Yaskawa INFORM job: DEMO_ROOF_SIDE_0625_3PAINT_40.JBI

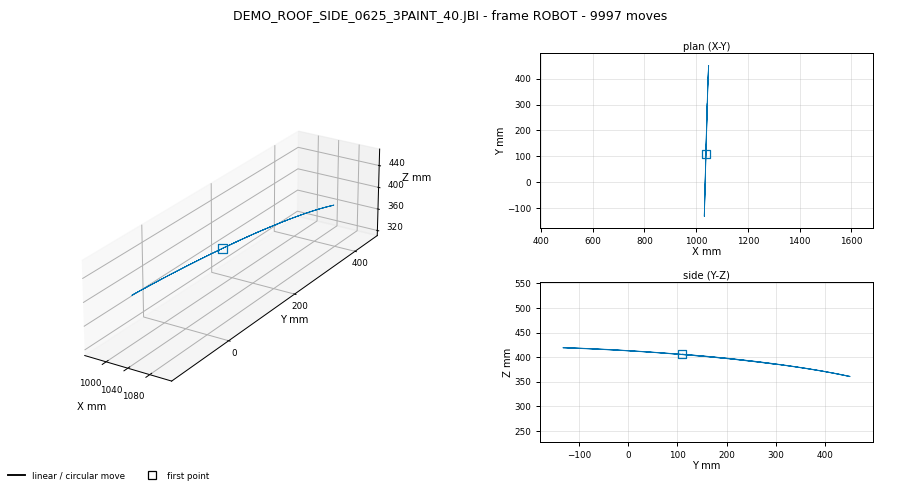
[picture p0: tool path of DEMO_ROOF_SIDE_0625_3PAINT_40.JBI in frame ROBOT, 9997 of 9997 moves have a stored position in this frame; points joined in program order, loops and branches not executed]
/JOB
//NAME DEMO_ROOF_SIDE_0625_3PAINT40
//POS
///NPOS 9997,0,0,0,0,0
///TOOL 0
///USER 0
///POSTYPE ROBOT
///RECTAN
///RCONF 1,0,0,0,0,0,0,0,0,0,0,0,0,0,0,0,0,0,0,0,0,0,0,0
C00000=1038.279,110.254,406.357,169.691,40.048,157.539
C00001=1038.285,110.504,406.337,169.693,40.048,157.539
C00002=1038.291,110.753,406.317,169.696,40.048,157.539
C00003=1038.297,111.002,406.297,169.698,40.048,157.539
C00004=1038.304,111.251,406.277,169.700,40.048,157.539
C00005=1038.310,111.500,406.257,169.702,40.049,157.539
C00006=1038.316,111.749,406.238,169.704,40.049,157.539
C00007=1038.323,111.998,406.218,169.706,40.049,157.539
C00008=1038.329,112.248,406.198,169.708,40.050,157.540
C00009=1038.335,112.497,406.178,169.710,40.049,157.540
C00010=1038.341,112.746,406.158,169.713,40.050,157.540
C00011=1038.347,112.995,406.138,169.715,40.050,157.540
C00012=1038.354,113.244,406.118,169.717,40.050,157.540
C00013=1038.359,113.494,406.097,169.719,40.051,157.540
C00014=1038.365,113.742,406.077,169.721,40.051,157.540
C00015=1038.372,113.992,406.057,169.723,40.051,157.540
C00016=1038.378,114.241,406.037,169.725,40.051,157.541
C00017=1038.383,114.490,406.016,169.727,40.052,157.541
C00018=1038.390,114.739,405.996,169.730,40.052,157.541
C00019=1038.396,114.988,405.976,169.732,40.052,157.541
C00020=1038.402,115.237,405.956,169.734,40.052,157.541
C00021=1038.407,115.487,405.935,169.736,40.053,157.541
C00022=1038.414,115.735,405.915,169.738,40.053,157.542
C00023=1038.420,115.984,405.895,169.740,40.053,157.542
C00024=1038.426,116.233,405.874,169.742,40.054,157.542
C00025=1038.432,116.482,405.854,169.745,40.054,157.542
C00026=1038.438,116.732,405.833,169.747,40.054,157.542
C00027=1038.444,116.981,405.813,169.749,40.054,157.542
C00028=1038.450,117.230,405.793,169.751,40.055,157.542
C00029=1038.456,117.479,405.773,169.753,40.055,157.543
C00030=1038.462,117.728,405.753,169.755,40.056,157.543
C00031=1038.469,117.977,405.732,169.757,40.055,157.543
C00032=1038.474,118.226,405.711,169.759,40.056,157.543
C00033=1038.480,118.475,405.691,169.762,40.056,157.543
C00034=1038.487,118.725,405.671,169.765,40.057,157.543
C00035=1038.493,118.973,405.651,169.767,40.057,157.543
C00036=1038.499,119.223,405.630,169.769,40.057,157.544
C00037=1038.505,119.471,405.609,169.771,40.057,157.544
C00038=1038.511,119.721,405.589,169.773,40.058,157.544
C00039=1038.517,119.970,405.569,169.775,40.058,157.544
C00040=1038.523,120.219,405.548,169.777,40.058,157.544
C00041=1038.529,120.468,405.528,169.780,40.059,157.544
C00042=1038.536,120.716,405.507,169.782,40.059,157.544
C00043=1038.541,120.966,405.486,169.784,40.059,157.544
C00044=1038.547,121.215,405.466,169.786,40.059,157.545
C00045=1038.554,121.465,405.446,169.788,40.060,157.545
C00046=1038.560,121.713,405.425,169.790,40.060,157.545
C00047=1038.566,121.963,405.404,169.792,40.060,157.545
C00048=1038.572,122.211,405.385,169.794,40.060,157.545
C00049=1038.579,122.460,405.363,169.797,40.061,157.545
C00050=1038.584,122.710,405.343,169.800,40.061,157.545
C00051=1038.591,122.959,405.323,169.802,40.061,157.546
C00052=1038.597,123.208,405.303,169.804,40.062,157.546
C00053=1038.603,123.457,405.281,169.806,40.061,157.546
C00054=1038.609,123.706,405.261,169.808,40.062,157.546
C00055=1038.616,123.955,405.241,169.810,40.062,157.546
C00056=1038.621,124.204,405.219,169.812,40.063,157.546
C00057=1038.628,124.453,405.199,169.814,40.062,157.546
C00058=1038.635,124.739,405.175,169.818,40.063,157.547
C00059=1038.642,125.025,405.151,169.820,40.063,157.547
C00060=1038.649,125.311,405.129,169.822,40.064,157.547
C00061=1038.656,125.596,405.105,169.825,40.064,157.547
C00062=1038.663,125.845,405.084,169.827,40.064,157.547
C00063=1038.668,126.094,405.063,169.829,40.064,157.547
C00064=1038.675,126.344,405.043,169.831,40.065,157.548
C00065=1038.682,126.593,405.022,169.833,40.065,157.548
C00066=1038.687,126.842,405.001,169.836,40.065,157.548
C00067=1038.694,127.091,404.980,169.838,40.065,157.548
C00068=1038.700,127.340,404.960,169.840,40.065,157.548
C00069=1038.706,127.589,404.939,169.843,40.066,157.548
C00070=1038.713,127.838,404.918,169.845,40.066,157.548
C00071=1038.719,128.086,404.898,169.847,40.067,157.549
C00072=1038.725,128.336,404.877,169.849,40.066,157.549
C00073=1038.731,128.585,404.857,169.851,40.067,157.549
C00074=1038.738,128.834,404.836,169.854,40.067,157.549
C00075=1038.744,129.084,404.815,169.856,40.067,157.549
C00076=1038.750,129.332,404.794,169.858,40.068,157.549
C00077=1038.757,129.582,404.774,169.861,40.068,157.549
C00078=1038.763,129.831,404.752,169.863,40.068,157.549
C00079=1038.769,130.080,404.732,169.865,40.068,157.550
C00080=1038.776,130.328,404.711,169.867,40.069,157.550
C00081=1038.782,130.578,404.690,169.869,40.068,157.550
C00082=1038.788,130.826,404.670,169.872,40.069,157.550
C00083=1038.795,131.075,404.649,169.874,40.069,157.550
C00084=1038.801,131.325,404.628,169.877,40.070,157.550
C00085=1038.806,131.574,404.606,169.879,40.070,157.551
C00086=1038.813,131.823,404.585,169.881,40.070,157.551
C00087=1038.818,132.072,404.565,169.883,40.070,157.551
C00088=1038.824,132.321,404.543,169.885,40.071,157.551
C00089=1038.831,132.570,404.522,169.888,40.071,157.551
C00090=1038.837,132.819,404.502,169.890,40.072,157.551
C00091=1038.843,133.068,404.480,169.892,40.072,157.551
C00092=1038.850,133.317,404.459,169.894,40.073,157.552
C00093=1038.855,133.566,404.438,169.896,40.072,157.552
C00094=1038.861,133.815,404.417,169.899,40.073,157.552
C00095=1038.868,134.064,404.396,169.901,40.073,157.552
C00096=1038.874,134.313,404.374,169.904,40.074,157.552
C00097=1038.879,134.563,404.354,169.906,40.074,157.552
C00098=1038.886,134.811,404.332,169.908,40.075,157.553
C00099=1038.892,135.060,404.311,169.910,40.074,157.553
C00100=1038.898,135.309,404.290,169.912,40.075,157.553
C00101=1038.905,135.559,404.269,169.914,40.075,157.553
C00102=1038.910,135.807,404.248,169.917,40.076,157.553
C00103=1038.916,136.056,404.226,169.920,40.076,157.553
C00104=1038.923,136.305,404.205,169.922,40.076,157.554
C00105=1038.928,136.554,404.185,169.924,40.076,157.554
C00106=1038.935,136.804,404.163,169.926,40.077,157.554
C00107=1038.942,137.053,404.142,169.928,40.077,157.554
C00108=1038.948,137.302,404.120,169.930,40.078,157.554
C00109=1038.953,137.550,404.099,169.933,40.078,157.554
C00110=1038.959,137.799,404.078,169.936,40.078,157.554
C00111=1038.966,138.048,404.056,169.938,40.079,157.555
C00112=1038.972,138.297,404.036,169.940,40.079,157.555
C00113=1038.978,138.547,404.014,169.942,40.079,157.555
C00114=1038.984,138.796,403.993,169.944,40.080,157.555
C00115=1038.991,139.045,403.972,169.947,40.080,157.555
C00116=1038.996,139.293,403.950,169.949,40.080,157.555
C00117=1039.003,139.542,403.929,169.952,40.081,157.556
C00118=1039.009,139.792,403.907,169.954,40.081,157.556
C00119=1039.015,140.041,403.885,169.956,40.082,157.556
C00120=1039.020,140.289,403.864,169.958,40.082,157.556
C00121=1039.027,140.539,403.843,169.960,40.083,157.556
C00122=1039.035,140.824,403.818,169.963,40.083,157.556
C00123=1039.041,141.110,403.794,169.966,40.083,157.557
C00124=1039.048,141.396,403.768,169.969,40.084,157.557
C00125=1039.055,141.681,403.745,169.971,40.084,157.557
C00126=1039.061,141.930,403.723,169.973,40.085,157.557
C00127=1039.067,142.179,403.701,169.976,40.085,157.557
C00128=1039.073,142.428,403.680,169.978,40.085,157.558
C00129=1039.079,142.676,403.658,169.981,40.086,157.558
C00130=1039.085,142.926,403.636,169.983,40.086,157.558
C00131=1039.092,143.175,403.614,169.985,40.087,157.558
C00132=1039.098,143.424,403.593,169.987,40.087,157.558
C00133=1039.103,143.673,403.571,169.990,40.088,157.558
C00134=1039.110,143.922,403.550,169.992,40.088,157.559
C00135=1039.116,144.171,403.528,169.995,40.088,157.559
C00136=1039.122,144.420,403.507,169.997,40.089,157.559
C00137=1039.129,144.669,403.486,169.999,40.089,157.559
C00138=1039.135,144.918,403.464,170.001,40.089,157.559
C00139=1039.141,145.166,403.442,170.004,40.089,157.559
C00140=1039.147,145.415,403.420,170.006,40.090,157.560
C00141=1039.153,145.665,403.399,170.008,40.090,157.560
C00142=1039.159,145.914,403.377,170.011,40.091,157.560
C00143=1039.165,146.163,403.355,170.013,40.091,157.560
C00144=1039.172,146.412,403.333,170.016,40.092,157.560
C00145=1039.178,146.661,403.311,170.018,40.092,157.560
C00146=1039.184,146.909,403.290,170.020,40.092,157.561
C00147=1039.190,147.159,403.268,170.022,40.093,157.561
C00148=1039.196,147.408,403.247,170.025,40.093,157.561
C00149=1039.202,147.656,403.225,170.028,40.094,157.561
C00150=1039.209,147.906,403.203,170.030,40.094,157.561
C00151=1039.215,148.155,403.181,170.032,40.095,157.562
C00152=1039.220,148.404,403.158,170.034,40.095,157.562
C00153=1039.226,148.652,403.137,170.036,40.095,157.562
C00154=1039.232,148.901,403.115,170.040,40.096,157.562
C00155=1039.238,149.151,403.094,170.042,40.096,157.562
C00156=1039.245,149.399,403.071,170.044,40.097,157.562
C00157=1039.251,149.648,403.050,170.046,40.097,157.563
C00158=1039.257,149.898,403.028,170.048,40.098,157.563
C00159=1039.263,150.146,403.005,170.051,40.098,157.563
C00160=1039.269,150.396,402.984,170.054,40.099,157.563
C00161=1039.276,150.644,402.961,170.056,40.099,157.563
C00162=1039.282,150.893,402.940,170.058,40.100,157.564
C00163=1039.287,151.142,402.918,170.060,40.100,157.564
C00164=1039.293,151.391,402.895,170.063,40.101,157.564
C00165=1039.299,151.640,402.874,170.066,40.101,157.564
C00166=1039.306,151.889,402.851,170.068,40.102,157.564
C00167=1039.312,152.138,402.830,170.070,40.102,157.565
C00168=1039.318,152.386,402.807,170.073,40.102,157.565
C00169=1039.324,152.636,402.785,170.075,40.103,157.565
C00170=1039.330,152.885,402.763,170.077,40.103,157.565
C00171=1039.336,153.134,402.741,170.079,40.104,157.565
C00172=1039.343,153.382,402.719,170.083,40.104,157.565
C00173=1039.349,153.632,402.697,170.085,40.104,157.566
C00174=1039.355,153.880,402.674,170.087,40.105,157.566
C00175=1039.361,154.130,402.653,170.089,40.106,157.566
C00176=1039.367,154.378,402.630,170.091,40.106,157.566
C00177=1039.373,154.627,402.609,170.095,40.107,157.567
C00178=1039.379,154.876,402.586,170.097,40.107,157.567
C00179=1039.385,155.126,402.564,170.099,40.108,157.567
C00180=1039.391,155.374,402.541,170.101,40.108,157.567
C00181=1039.397,155.624,402.519,170.104,40.108,157.567
C00182=1039.404,155.872,402.497,170.107,40.109,157.568
C00183=1039.409,156.121,402.474,170.109,40.110,157.568
C00184=1039.416,156.370,402.453,170.111,40.110,157.568
C00185=1039.422,156.619,402.430,170.114,40.111,157.568
C00186=1039.429,156.904,402.405,170.116,40.111,157.568
C00187=1039.435,157.189,402.379,170.120,40.112,157.569
C00188=1039.442,157.475,402.354,170.122,40.113,157.569
C00189=1039.449,157.760,402.328,170.125,40.113,157.569
C00190=1039.456,158.009,402.306,170.127,40.113,157.569
C00191=1039.462,158.257,402.284,170.130,40.114,157.569
C00192=1039.468,158.506,402.261,170.133,40.115,157.570
C00193=1039.474,158.755,402.238,170.135,40.115,157.570
C00194=1039.480,159.004,402.216,170.137,40.116,157.570
C00195=1039.486,159.253,402.194,170.140,40.116,157.570
C00196=1039.493,159.502,402.171,170.142,40.116,157.570
C00197=1039.498,159.751,402.148,170.144,40.117,157.571
C00198=1039.505,160.000,402.126,170.147,40.118,157.571
C00199=1039.511,160.249,402.103,170.150,40.118,157.571
C00200=1039.517,160.498,402.081,170.152,40.119,157.571
C00201=1039.523,160.747,402.058,170.154,40.120,157.572
C00202=1039.529,160.996,402.035,170.157,40.120,157.572
C00203=1039.535,161.245,402.012,170.160,40.121,157.572
C00204=1039.540,161.494,401.990,170.162,40.122,157.572
C00205=1039.546,161.743,401.968,170.164,40.122,157.572
C00206=1039.552,161.992,401.945,170.166,40.122,157.573
C00207=1039.558,162.241,401.922,170.170,40.123,157.573
C00208=1039.564,162.489,401.899,170.172,40.124,157.573
C00209=1039.570,162.738,401.876,170.174,40.124,157.573
C00210=1039.576,162.987,401.854,170.176,40.125,157.574
C00211=1039.582,163.236,401.831,170.179,40.126,157.574
C00212=1039.587,163.485,401.808,170.182,40.127,157.574
C00213=1039.593,163.734,401.785,170.184,40.127,157.574
C00214=1039.599,163.982,401.762,170.187,40.128,157.574
C00215=1039.605,164.231,401.739,170.189,40.129,157.575
C00216=1039.611,164.480,401.716,170.192,40.129,157.575
C00217=1039.617,164.729,401.694,170.194,40.130,157.575
C00218=1039.623,164.978,401.670,170.197,40.131,157.575
C00219=1039.629,165.227,401.648,170.199,40.131,157.576
C00220=1039.635,165.476,401.625,170.202,40.132,157.576
C00221=1039.641,165.725,401.602,170.204,40.132,157.576
C00222=1039.647,165.974,401.579,170.207,40.133,157.576
C00223=1039.652,166.223,401.556,170.209,40.134,157.577
C00224=1039.659,166.471,401.533,170.211,40.134,157.577
C00225=1039.665,166.719,401.510,170.215,40.135,157.577
C00226=1039.671,166.969,401.487,170.217,40.136,157.577
C00227=1039.677,167.218,401.464,170.219,40.136,157.577
C00228=1039.683,167.467,401.441,170.222,40.137,157.578
C00229=1039.689,167.715,401.418,170.224,40.138,157.578
C00230=1039.695,167.964,401.396,170.227,40.139,157.578
C00231=1039.701,168.213,401.373,170.230,40.139,157.579
C00232=1039.707,168.462,401.349,170.232,40.139,157.579
C00233=1039.713,168.711,401.326,170.234,40.140,157.579
C00234=1039.719,168.960,401.303,170.238,40.141,157.579
C00235=1039.725,169.209,401.280,170.240,40.142,157.579
C00236=1039.731,169.458,401.257,170.242,40.142,157.580
C00237=1039.737,169.706,401.234,170.245,40.143,157.580
C00238=1039.743,169.955,401.210,170.248,40.144,157.580
C00239=1039.749,170.204,401.187,170.250,40.144,157.580
C00240=1039.756,170.453,401.165,170.253,40.145,157.581
C00241=1039.761,170.702,401.142,170.255,40.146,157.581
C00242=1039.768,170.951,401.118,170.257,40.146,157.581
C00243=1039.774,171.200,401.095,170.261,40.147,157.581
C00244=1039.779,171.449,401.072,170.263,40.147,157.582
C00245=1039.785,171.697,401.049,170.265,40.148,157.582
C00246=1039.792,171.946,401.025,170.268,40.149,157.582
C00247=1039.798,172.195,401.003,170.271,40.149,157.582
C00248=1039.804,172.444,400.980,170.273,40.150,157.583
C00249=1039.810,172.692,400.956,170.276,40.151,157.583
C00250=1039.817,172.978,400.930,170.279,40.152,157.583
C00251=1039.824,173.262,400.903,170.282,40.152,157.583
C00252=1039.831,173.547,400.877,170.285,40.153,157.584
C00253=1039.838,173.831,400.850,170.288,40.154,157.584
C00254=1039.844,174.080,400.827,170.290,40.154,157.584
C00255=1039.850,174.330,400.804,170.294,40.155,157.584
C00256=1039.857,174.578,400.780,170.296,40.156,157.585
C00257=1039.862,174.827,400.757,170.298,40.156,157.585
C00258=1039.869,175.076,400.733,170.301,40.157,157.585
C00259=1039.875,175.325,400.711,170.303,40.158,157.585
C00260=1039.881,175.574,400.688,170.307,40.159,157.586
C00261=1039.888,175.823,400.664,170.309,40.159,157.586
C00262=1039.893,176.071,400.641,170.311,40.160,157.586
C00263=1039.899,176.320,400.617,170.314,40.160,157.586
C00264=1039.906,176.569,400.594,170.317,40.161,157.587
C00265=1039.912,176.818,400.570,170.320,40.162,157.587
C00266=1039.918,177.067,400.547,170.322,40.162,157.587
C00267=1039.925,177.315,400.524,170.324,40.163,157.587
C00268=1039.931,177.564,400.501,170.328,40.164,157.587
C00269=1039.937,177.813,400.477,170.330,40.165,157.588
C00270=1039.943,178.062,400.454,170.333,40.165,157.588
C00271=1039.949,178.310,400.430,170.335,40.166,157.588
C00272=1039.955,178.560,400.407,170.339,40.166,157.589
C00273=1039.961,178.808,400.383,170.341,40.168,157.589
C00274=1039.968,179.058,400.360,170.344,40.168,157.589
C00275=1039.974,179.306,400.336,170.346,40.169,157.589
C00276=1039.981,179.555,400.313,170.350,40.169,157.590
C00277=1039.987,179.804,400.290,170.352,40.170,157.590
C00278=1039.994,180.053,400.266,170.354,40.171,157.590
C00279=1039.999,180.301,400.243,170.357,40.171,157.590
C00280=1040.005,180.550,400.219,170.359,40.172,157.591
C00281=1040.012,180.799,400.195,170.363,40.172,157.591
C00282=1040.018,181.048,400.172,170.365,40.174,157.591
C00283=1040.024,181.297,400.148,170.368,40.174,157.591
C00284=1040.030,181.545,400.124,170.370,40.175,157.592
C00285=1040.037,181.794,400.101,170.374,40.175,157.592
C00286=1040.044,182.042,400.078,170.376,40.176,157.592
C00287=1040.050,182.291,400.054,170.379,40.177,157.592
C00288=1040.056,182.540,400.031,170.381,40.178,157.593
C00289=1040.063,182.789,400.007,170.385,40.178,157.593
C00290=1040.069,183.038,399.983,170.387,40.179,157.593
C00291=1040.075,183.287,399.959,170.390,40.179,157.593
C00292=1040.082,183.536,399.936,170.392,40.180,157.594
C00293=1040.087,183.785,399.912,170.396,40.181,157.594
C00294=1040.093,184.034,399.888,170.398,40.182,157.594
C00295=1040.099,184.282,399.864,170.401,40.183,157.594
C00296=1040.105,184.531,399.840,170.404,40.184,157.595
C00297=1040.111,184.780,399.816,170.406,40.185,157.595
C00298=1040.117,185.028,399.792,170.409,40.186,157.595
C00299=1040.123,185.277,399.768,170.411,40.186,157.596
C00300=1040.129,185.526,399.743,170.415,40.187,157.596
C00301=1040.135,185.775,399.719,170.417,40.188,157.596
C00302=1040.141,186.023,399.695,170.420,40.189,157.597
C00303=1040.147,186.272,399.671,170.423,40.190,157.597
C00304=1040.153,186.521,399.647,170.426,40.191,157.597
C00305=1040.159,186.770,399.623,170.428,40.192,157.597
C00306=1040.164,187.018,399.598,170.431,40.193,157.598
C00307=1040.171,187.267,399.574,170.434,40.194,157.598
C00308=1040.176,187.516,399.550,170.437,40.195,157.598
C00309=1040.183,187.765,399.526,170.439,40.196,157.599
C00310=1040.188,188.014,399.502,170.443,40.196,157.599
C00311=1040.195,188.262,399.478,170.445,40.197,157.599
C00312=1040.200,188.511,399.454,170.448,40.198,157.599
C00313=1040.207,188.760,399.430,170.450,40.199,157.600
C00314=1040.214,189.044,399.402,170.454,40.200,157.600
C00315=1040.221,189.328,399.375,170.457,40.201,157.600
C00316=1040.227,189.613,399.346,170.460,40.202,157.601
C00317=1040.234,189.897,399.319,170.463,40.203,157.601
C00318=1040.240,190.146,399.295,170.466,40.204,157.601
C00319=1040.247,190.395,399.270,170.469,40.205,157.602
C00320=1040.253,190.643,399.246,170.472,40.206,157.602
C00321=1040.259,190.892,399.221,170.475,40.207,157.602
C00322=1040.265,191.141,399.198,170.477,40.208,157.603
C00323=1040.271,191.390,399.173,170.481,40.209,157.603
C00324=1040.277,191.638,399.148,170.483,40.209,157.603
C00325=1040.283,191.887,399.124,170.486,40.210,157.604
C00326=1040.289,192.136,399.100,170.488,40.211,157.604
C00327=1040.295,192.385,399.075,170.492,40.212,157.604
C00328=1040.302,192.633,399.051,170.494,40.213,157.605
C00329=1040.308,192.882,399.026,170.497,40.214,157.605
C00330=1040.313,193.131,399.002,170.500,40.215,157.605
C00331=1040.319,193.380,398.978,170.503,40.216,157.606
C00332=1040.326,193.628,398.953,170.506,40.217,157.606
C00333=1040.332,193.877,398.929,170.509,40.218,157.606
C00334=1040.338,194.126,398.904,170.512,40.219,157.606
C00335=1040.345,194.374,398.880,170.514,40.220,157.607
C00336=1040.350,194.623,398.855,170.518,40.221,157.607
C00337=1040.357,194.872,398.831,170.520,40.222,157.607
C00338=1040.363,195.120,398.806,170.523,40.223,157.608
C00339=1040.369,195.369,398.782,170.527,40.224,157.608
C00340=1040.375,195.617,398.757,170.529,40.225,157.608
C00341=1040.381,195.867,398.732,170.532,40.226,157.609
C00342=1040.387,196.116,398.708,170.534,40.227,157.609
C00343=1040.394,196.364,398.683,170.538,40.228,157.609
C00344=1040.400,196.613,398.659,170.541,40.229,157.610
C00345=1040.406,196.861,398.634,170.543,40.230,157.610
C00346=1040.413,197.110,398.610,170.547,40.231,157.610
C00347=1040.419,197.359,398.585,170.549,40.232,157.611
C00348=1040.425,197.608,398.561,170.552,40.233,157.611
C00349=1040.431,197.856,398.536,170.556,40.233,157.611
C00350=1040.437,198.105,398.511,170.558,40.234,157.611
C00351=1040.444,198.353,398.486,170.561,40.235,157.612
C00352=1040.450,198.603,398.462,170.565,40.236,157.612
C00353=1040.457,198.851,398.437,170.567,40.237,157.612
C00354=1040.462,199.100,398.413,170.570,40.238,157.613
C00355=1040.469,199.348,398.388,170.572,40.239,157.613
C00356=1040.475,199.597,398.363,170.576,40.240,157.613
C00357=1040.481,199.846,398.338,170.579,40.241,157.614
C00358=1040.488,200.095,398.314,170.581,40.242,157.614
C00359=1040.494,200.344,398.289,170.585,40.243,157.614
C00360=1040.500,200.591,398.264,170.588,40.244,157.615
C00361=1040.506,200.841,398.240,170.590,40.245,157.615
C00362=1040.512,201.089,398.214,170.594,40.246,157.615
C00363=1040.519,201.338,398.189,170.597,40.247,157.616
C00364=1040.525,201.587,398.165,170.600,40.248,157.616
C00365=1040.531,201.836,398.140,170.603,40.249,157.616
C00366=1040.537,202.084,398.115,170.606,40.250,157.617
C00367=1040.543,202.333,398.090,170.609,40.251,157.617
C00368=1040.549,202.582,398.065,170.612,40.253,157.618
C00369=1040.555,202.830,398.039,170.614,40.254,157.618
C00370=1040.562,203.079,398.014,170.618,40.255,157.618
C00371=1040.568,203.328,397.989,170.621,40.256,157.619
C00372=1040.574,203.577,397.964,170.623,40.257,157.619
C00373=1040.579,203.825,397.939,170.627,40.259,157.619
C00374=1040.585,204.073,397.914,170.630,40.259,157.620
C00375=1040.592,204.322,397.888,170.632,40.261,157.620
C00376=1040.599,204.571,397.864,170.636,40.261,157.620
C00377=1040.605,204.819,397.838,170.639,40.263,157.621
C00378=1040.631,205.871,397.732,170.925,40.366,157.654
C00379=1040.639,206.173,397.700,170.927,40.368,157.655
C00380=1040.647,206.477,397.667,170.930,40.370,157.656
C00381=1040.655,206.780,397.635,170.933,40.373,157.656
C00382=1040.664,207.084,397.604,170.935,40.375,157.657
C00383=1040.670,207.333,397.577,170.938,40.377,157.657
C00384=1040.677,207.581,397.551,170.939,40.379,157.658
C00385=1040.684,207.830,397.524,170.942,40.380,157.658
C00386=1040.689,208.078,397.498,170.944,40.383,157.659
C00387=1040.697,208.326,397.470,170.946,40.384,157.659
C00388=1040.703,208.574,397.444,170.948,40.386,157.660
C00389=1040.710,208.823,397.417,170.951,40.388,157.660
C00390=1040.717,209.072,397.391,170.952,40.390,157.661
C00391=1040.723,209.320,397.365,170.955,40.392,157.661
C00392=1040.730,209.569,397.338,170.957,40.393,157.662
C00393=1040.736,209.817,397.312,170.959,40.396,157.662
C00394=1040.743,210.066,397.285,170.962,40.397,157.663
C00395=1040.750,210.315,397.258,170.964,40.399,157.663
C00396=1040.757,210.562,397.232,170.967,40.401,157.664
C00397=1040.764,210.811,397.205,170.968,40.403,157.664
C00398=1040.769,211.059,397.179,170.971,40.405,157.665
C00399=1040.777,211.308,397.152,170.973,40.407,157.665
C00400=1040.783,211.557,397.125,170.976,40.409,157.666
C00401=1040.790,211.805,397.098,170.977,40.410,157.666
C00402=1040.796,212.054,397.071,170.980,40.413,157.667
C00403=1040.803,212.302,397.045,170.982,40.414,157.667
C00404=1040.809,212.551,397.018,170.984,40.416,157.668
C00405=1040.816,212.799,396.991,170.986,40.418,157.668
C00406=1040.822,213.047,396.965,170.989,40.420,157.669
C00407=1040.829,213.296,396.938,170.991,40.422,157.669
C00408=1040.836,213.544,396.910,170.993,40.424,157.670
C00409=1040.843,213.792,396.884,170.995,40.426,157.670
C00410=1040.849,214.042,396.857,170.998,40.428,157.671
C00411=1040.856,214.290,396.830,171.001,40.430,157.671
C00412=1040.862,214.538,396.804,171.002,40.431,157.672
C00413=1040.868,214.787,396.777,171.005,40.434,157.672
C00414=1040.876,215.035,396.749,171.007,40.435,157.673
C00415=1040.882,215.284,396.723,171.010,40.437,157.673
C00416=1040.889,215.532,396.696,171.012,40.439,157.674
C00417=1040.895,215.781,396.669,171.014,40.441,157.674
C00418=1040.903,216.030,396.642,171.016,40.443,157.675
C00419=1040.909,216.277,396.615,171.019,40.444,157.675
C00420=1040.915,216.526,396.588,171.021,40.446,157.676
C00421=1040.922,216.775,396.561,171.023,40.448,157.676
C00422=1040.928,217.023,396.534,171.025,40.450,157.676
C00423=1040.935,217.272,396.508,171.028,40.452,157.677
C00424=1040.942,217.520,396.480,171.030,40.454,157.678
C00425=1040.949,217.769,396.453,171.033,40.455,157.678
C00426=1040.955,218.017,396.426,171.035,40.458,157.679
C00427=1040.962,218.266,396.399,171.037,40.459,157.679
C00428=1040.969,218.514,396.372,171.040,40.461,157.679
C00429=1040.975,218.763,396.345,171.042,40.463,157.680
C00430=1040.982,219.010,396.318,171.045,40.465,157.681
C00431=1040.989,219.259,396.291,171.047,40.467,157.681
C00432=1040.996,219.507,396.264,171.049,40.468,157.681
C00433=1041.002,219.756,396.237,171.051,40.471,157.682
C00434=1041.009,220.005,396.209,171.054,40.472,157.682
C00435=1041.018,220.313,396.176,171.056,40.474,157.683
C00436=1041.025,220.622,396.142,171.060,40.477,157.684
C00437=1041.033,220.931,396.108,171.063,40.479,157.684
C00438=1041.042,221.240,396.074,171.065,40.482,157.685
C00439=1041.049,221.488,396.046,171.068,40.483,157.685
C00440=1041.055,221.737,396.019,171.071,40.486,157.686
C00441=1041.061,221.985,395.992,171.073,40.487,157.687
C00442=1041.068,222.233,395.964,171.076,40.489,157.687
C00443=1041.075,222.482,395.938,171.077,40.491,157.688
C00444=1041.081,222.730,395.910,171.080,40.493,157.688
C00445=1041.088,222.979,395.882,171.082,40.495,157.688
C00446=1041.094,223.227,395.855,171.085,40.497,157.689
C00447=1041.101,223.476,395.828,171.087,40.498,157.690
C00448=1041.107,223.724,395.800,171.090,40.500,157.690
C00449=1041.114,223.973,395.773,171.092,40.502,157.691
C00450=1041.121,224.221,395.745,171.094,40.504,157.691
C00451=1041.128,224.470,395.718,171.097,40.506,157.692
C00452=1041.134,224.718,395.691,171.099,40.508,157.692
C00453=1041.141,224.966,395.663,171.101,40.510,157.693
C00454=1041.147,225.214,395.636,171.104,40.512,157.693
C00455=1041.154,225.463,395.608,171.107,40.513,157.694
C00456=1041.161,225.711,395.580,171.109,40.515,157.694
C00457=1041.168,225.960,395.554,171.112,40.517,157.695
C00458=1041.174,226.209,395.526,171.114,40.519,157.695
C00459=1041.180,226.456,395.499,171.116,40.521,157.696
C00460=1041.187,226.705,395.471,171.118,40.523,157.696
C00461=1041.194,226.953,395.443,171.121,40.525,157.697
C00462=1041.200,227.202,395.415,171.123,40.526,157.697
C00463=1041.207,227.450,395.388,171.126,40.529,157.698
C00464=1041.214,227.698,395.360,171.128,40.530,157.698
C00465=1041.221,227.947,395.332,171.131,40.532,157.699
C00466=1041.228,228.196,395.306,171.134,40.534,157.699
C00467=1041.234,228.444,395.278,171.136,40.536,157.700
C00468=1041.241,228.693,395.250,171.139,40.537,157.700
C00469=1041.248,228.941,395.223,171.141,40.540,157.701
C00470=1041.254,229.190,395.194,171.144,40.541,157.701
C00471=1041.260,229.437,395.166,171.146,40.543,157.702
C00472=1041.267,229.685,395.138,171.149,40.545,157.702
C00473=1041.273,229.934,395.111,171.150,40.547,157.703
C00474=1041.280,230.182,395.083,171.153,40.549,157.703
C00475=1041.287,230.431,395.055,171.155,40.551,157.704
C00476=1041.293,230.679,395.028,171.158,40.553,157.704
C00477=1041.300,230.927,395.000,171.161,40.555,157.705
C00478=1041.307,231.176,394.972,171.163,40.556,157.705
C00479=1041.313,231.424,394.944,171.166,40.558,157.706
C00480=1041.319,231.673,394.916,171.168,40.560,157.706
C00481=1041.326,231.921,394.888,171.171,40.562,157.707
C00482=1041.333,232.169,394.860,171.173,40.564,157.707
C00483=1041.340,232.418,394.832,171.176,40.566,157.708
C00484=1041.346,232.666,394.804,171.179,40.568,157.708
C00485=1041.352,232.915,394.776,171.181,40.569,157.709
C00486=1041.359,233.163,394.748,171.184,40.572,157.709
C00487=1041.366,233.411,394.720,171.186,40.573,157.710
C00488=1041.373,233.660,394.692,171.189,40.576,157.710
C00489=1041.379,233.908,394.664,171.191,40.577,157.711
C00490=1041.386,234.156,394.635,171.194,40.579,157.712
C00491=1041.393,234.457,394.602,171.197,40.582,157.712
C00492=1041.401,234.759,394.568,171.200,40.584,157.713
C00493=1041.410,235.060,394.534,171.203,40.586,157.713
C00494=1041.418,235.362,394.499,171.206,40.588,157.714
C00495=1041.424,235.610,394.471,171.208,40.590,157.715
C00496=1041.431,235.858,394.444,171.211,40.592,157.715
C00497=1041.437,236.107,394.415,171.213,40.594,157.715
C00498=1041.444,236.355,394.387,171.217,40.596,157.716
C00499=1041.451,236.603,394.359,171.219,40.597,157.717
C00500=1041.457,236.852,394.330,171.222,40.600,157.717
C00501=1041.464,237.100,394.302,171.224,40.601,157.718
C00502=1041.471,237.348,394.274,171.227,40.604,157.718
C00503=1041.477,237.596,394.246,171.230,40.605,157.719
C00504=1041.483,237.845,394.218,171.232,40.607,157.719
C00505=1041.490,238.093,394.189,171.235,40.609,157.720
C00506=1041.497,238.342,394.161,171.237,40.611,157.720
C00507=1041.504,238.590,394.132,171.240,40.613,157.721
C00508=1041.510,238.839,394.105,171.242,40.615,157.721
C00509=1041.517,239.086,394.076,171.245,40.617,157.722
C00510=1041.523,239.335,394.048,171.248,40.618,157.722
C00511=1041.530,239.583,394.019,171.250,40.620,157.723
C00512=1041.537,239.831,393.992,171.253,40.622,157.723
C00513=1041.543,240.080,393.963,171.255,40.624,157.724
C00514=1041.550,240.328,393.935,171.258,40.626,157.724
C00515=1041.557,240.577,393.906,171.260,40.628,157.725
C00516=1041.563,240.825,393.878,171.263,40.630,157.726
C00517=1041.570,241.073,393.849,171.267,40.631,157.726
C00518=1041.577,241.321,393.820,171.269,40.634,157.727
C00519=1041.583,241.570,393.793,171.272,40.635,157.727
C00520=1041.590,241.818,393.763,171.274,40.638,157.728
C00521=1041.596,242.066,393.734,171.277,40.639,157.728
C00522=1041.603,242.315,393.706,171.279,40.641,157.729
C00523=1041.609,242.563,393.677,171.282,40.643,157.729
C00524=1041.616,242.811,393.649,171.285,40.645,157.730
C00525=1041.623,243.059,393.620,171.287,40.647,157.730
C00526=1041.629,243.308,393.592,171.290,40.649,157.731
C00527=1041.636,243.556,393.563,171.292,40.651,157.731
C00528=1041.642,243.804,393.534,171.295,40.653,157.732
C00529=1041.649,244.052,393.505,171.297,40.655,157.732
C00530=1041.655,244.301,393.477,171.301,40.657,157.733
C00531=1041.662,244.549,393.448,171.304,40.658,157.733
C00532=1041.669,244.797,393.419,171.306,40.660,157.734
C00533=1041.675,245.045,393.390,171.309,40.662,157.735
C00534=1041.682,245.294,393.362,171.311,40.664,157.735
C00535=1041.688,245.543,393.333,171.314,40.667,157.736
C00536=1041.695,245.791,393.304,171.317,40.668,157.736
C00537=1041.701,246.039,393.275,171.319,40.670,157.737
C00538=1041.707,246.287,393.246,171.322,40.672,157.737
C00539=1041.713,246.535,393.217,171.325,40.674,157.738
C00540=1041.721,246.784,393.188,171.328,40.676,157.739
C00541=1041.727,247.032,393.159,171.331,40.678,157.739
C00542=1041.733,247.280,393.130,171.333,40.680,157.740
C00543=1041.740,247.528,393.101,171.336,40.682,157.740
C00544=1041.746,247.776,393.072,171.338,40.684,157.741
C00545=1041.753,248.025,393.043,171.341,40.686,157.741
C00546=1041.759,248.273,393.014,171.344,40.688,157.742
C00547=1041.767,248.569,392.979,171.347,40.691,157.742
C00548=1041.774,248.864,392.945,171.351,40.693,157.743
C00549=1041.783,249.160,392.910,171.354,40.695,157.744
C00550=1041.791,249.455,392.875,171.358,40.698,157.744
C00551=1041.797,249.703,392.846,171.360,40.699,157.745
C00552=1041.803,249.951,392.817,171.363,40.701,157.746
C00553=1041.809,250.199,392.788,171.365,40.704,157.746
C00554=1041.816,250.448,392.759,171.368,40.705,157.747
C00555=1041.823,250.696,392.730,171.372,40.707,157.747
C00556=1041.830,250.944,392.701,171.374,40.709,157.748
C00557=1041.837,251.192,392.671,171.377,40.711,157.748
C00558=1041.843,251.441,392.642,171.379,40.713,157.749
C00559=1041.849,251.689,392.613,171.382,40.715,157.749
C00560=1041.856,251.938,392.584,171.386,40.717,157.750
C00561=1041.862,252.186,392.555,171.388,40.719,157.750
C00562=1041.869,252.433,392.525,171.391,40.721,157.751
C00563=1041.876,252.682,392.496,171.393,40.723,157.752
C00564=1041.882,252.930,392.466,171.396,40.725,157.752
C00565=1041.889,253.178,392.438,171.400,40.727,157.753
C00566=1041.896,253.427,392.409,171.402,40.729,157.753
C00567=1041.902,253.674,392.379,171.405,40.731,157.754
C00568=1041.909,253.922,392.350,171.407,40.733,157.754
C00569=1041.915,254.171,392.320,171.410,40.735,157.755
C00570=1041.922,254.419,392.291,171.414,40.737,157.756
C00571=1041.929,254.668,392.261,171.416,40.739,157.756
C00572=1041.935,254.916,392.232,171.419,40.741,157.757
C00573=1041.941,255.164,392.203,171.421,40.743,157.757
C00574=1041.949,255.412,392.173,171.425,40.744,157.758
C00575=1041.955,255.660,392.144,171.428,40.746,157.758
C00576=1041.963,255.908,392.114,171.430,40.749,157.759
C00577=1041.969,256.156,392.085,171.434,40.750,157.759
C00578=1041.975,256.404,392.056,171.436,40.752,157.760
C00579=1041.982,256.653,392.026,171.439,40.754,157.761
C00580=1041.989,256.901,391.997,171.442,40.756,157.761
C00581=1041.996,257.149,391.967,171.445,40.758,157.762
C00582=1042.002,257.397,391.938,171.448,40.760,157.762
C00583=1042.009,257.646,391.909,171.450,40.762,157.763
C00584=1042.015,257.893,391.879,171.454,40.764,157.763
C00585=1042.022,258.142,391.850,171.457,40.766,157.764
C00586=1042.029,258.390,391.820,171.459,40.768,157.765
C00587=1042.036,258.639,391.790,171.462,40.770,157.765
C00588=1042.042,258.886,391.761,171.465,40.772,157.766
C00589=1042.050,259.135,391.732,171.468,40.774,157.766
C00590=1042.056,259.382,391.702,171.471,40.776,157.767
C00591=1042.063,259.631,391.673,171.474,40.778,157.767
C00592=1042.070,259.878,391.643,171.477,40.779,157.768
C00593=1042.077,260.127,391.613,171.479,40.781,157.768
C00594=1042.084,260.376,391.583,171.483,40.784,157.769
C00595=1042.090,260.623,391.554,171.486,40.785,157.770
C00596=1042.097,260.872,391.524,171.488,40.787,157.770
C00597=1042.104,261.119,391.494,171.492,40.789,157.771
C00598=1042.111,261.368,391.465,171.495,40.791,157.771
C00599=1042.117,261.616,391.435,171.497,40.793,157.772
C00600=1042.124,261.864,391.405,171.501,40.795,157.772
C00601=1042.131,262.113,391.376,171.503,40.797,157.773
C00602=1042.138,262.360,391.346,171.507,40.799,157.774
C00603=1042.146,262.654,391.311,171.510,40.801,157.774
C00604=1042.153,262.948,391.274,171.514,40.804,157.775
C00605=1042.161,263.243,391.239,171.517,40.806,157.776
C00606=1042.169,263.537,391.204,171.521,40.809,157.776
C00607=1042.176,263.785,391.174,171.524,40.811,157.777
C00608=1042.182,264.033,391.143,171.526,40.812,157.777
C00609=1042.189,264.281,391.113,171.530,40.815,157.778
C00610=1042.195,264.528,391.084,171.533,40.817,157.779
C00611=1042.202,264.778,391.054,171.535,40.819,157.779
C00612=1042.209,265.026,391.023,171.539,40.821,157.780
C00613=1042.215,265.273,390.994,171.541,40.823,157.780
C00614=1042.222,265.522,390.963,171.545,40.825,157.781
C00615=1042.228,265.769,390.933,171.548,40.827,157.782
C00616=1042.235,266.018,390.903,171.551,40.829,157.782
C00617=1042.242,266.266,390.872,171.554,40.831,157.783
C00618=1042.248,266.514,390.843,171.557,40.833,157.783
C00619=1042.255,266.762,390.812,171.559,40.835,157.784
C00620=1042.262,267.010,390.782,171.563,40.837,157.785
C00621=1042.268,267.258,390.752,171.566,40.839,157.785
C00622=1042.276,267.506,390.722,171.569,40.841,157.786
C00623=1042.282,267.755,390.691,171.572,40.844,157.786
C00624=1042.289,268.002,390.661,171.575,40.845,157.787
C00625=1042.295,268.251,390.631,171.578,40.847,157.788
C00626=1042.302,268.499,390.601,171.581,40.849,157.788
C00627=1042.308,268.747,390.570,171.585,40.852,157.789
C00628=1042.315,268.995,390.540,171.587,40.854,157.789
C00629=1042.322,269.243,390.509,171.591,40.856,157.790
C00630=1042.328,269.490,390.479,171.594,40.858,157.791
C00631=1042.335,269.739,390.448,171.596,40.860,157.791
C00632=1042.342,269.987,390.418,171.600,40.862,157.792
C00633=1042.348,270.235,390.388,171.603,40.864,157.792
C00634=1042.355,270.483,390.358,171.606,40.866,157.793
C00635=1042.362,270.731,390.326,171.609,40.868,157.794
C00636=1042.368,270.978,390.296,171.613,40.870,157.794
C00637=1042.375,271.227,390.266,171.615,40.872,157.795
C00638=1042.382,271.475,390.236,171.619,40.875,157.796
C00639=1042.389,271.723,390.204,171.622,40.877,157.796
C00640=1042.394,271.971,390.174,171.624,40.879,157.797
C00641=1042.402,272.219,390.144,171.628,40.881,157.797
C00642=1042.408,272.467,390.112,171.631,40.883,157.798
C00643=1042.415,272.715,390.082,171.634,40.885,157.799
C00644=1042.421,272.963,390.052,171.637,40.887,157.799
C00645=1042.428,273.211,390.020,171.641,40.889,157.800
C00646=1042.435,273.459,389.990,171.643,40.891,157.800
C00647=1042.442,273.708,389.959,171.647,40.893,157.801
C00648=1042.448,273.955,389.928,171.650,40.895,157.802
C00649=1042.455,274.203,389.898,171.653,40.897,157.802
C00650=1042.462,274.451,389.867,171.656,40.900,157.803
C00651=1042.468,274.700,389.836,171.660,40.902,157.804
C00652=1042.475,274.947,389.805,171.662,40.904,157.804
C00653=1042.481,275.195,389.775,171.666,40.906,157.805
C00654=1042.488,275.443,389.744,171.669,40.908,157.805
C00655=1042.494,275.691,389.713,171.672,40.910,157.806
C00656=1042.502,275.939,389.682,171.675,40.912,157.807
C00657=1042.508,276.188,389.651,171.679,40.914,157.807
C00658=1042.514,276.435,389.620,171.682,40.917,157.808
C00659=1042.523,276.733,389.583,171.685,40.919,157.809
C00660=1042.530,277.032,389.546,171.689,40.922,157.809
C00661=1042.539,277.331,389.509,171.693,40.925,157.810
C00662=1042.547,277.630,389.471,171.697,40.927,157.811
C00663=1042.553,277.877,389.440,171.701,40.929,157.812
C00664=1042.560,278.125,389.410,171.704,40.931,157.812
C00665=1042.567,278.373,389.378,171.707,40.934,157.813
C00666=1042.574,278.621,389.347,171.711,40.936,157.814
C00667=1042.580,278.870,389.316,171.713,40.938,157.814
C00668=1042.587,279.117,389.285,171.717,40.940,157.815
C00669=1042.594,279.365,389.253,171.720,40.942,157.815
C00670=1042.600,279.613,389.222,171.724,40.945,157.816
C00671=1042.606,279.861,389.191,171.726,40.947,157.817
C00672=1042.613,280.109,389.160,171.730,40.949,157.817
C00673=1042.620,280.357,389.129,171.734,40.951,157.818
C00674=1042.626,280.605,389.097,171.736,40.953,157.819
C00675=1042.633,280.853,389.066,171.740,40.955,157.819
C00676=1042.640,281.101,389.035,171.743,40.958,157.820
C00677=1042.646,281.349,389.004,171.747,40.960,157.821
C00678=1042.653,281.597,388.972,171.749,40.962,157.821
C00679=1042.660,281.845,388.941,171.753,40.964,157.822
C00680=1042.666,282.093,388.909,171.757,40.967,157.823
C00681=1042.673,282.341,388.878,171.760,40.969,157.823
C00682=1042.680,282.589,388.846,171.763,40.971,157.824
C00683=1042.687,282.837,388.815,171.766,40.974,157.825
C00684=1042.693,283.084,388.784,171.770,40.976,157.825
C00685=1042.700,283.332,388.752,171.773,40.978,157.826
C00686=1042.707,283.580,388.721,171.776,40.980,157.827
C00687=1042.714,283.828,388.689,171.780,40.983,157.827
C00688=1042.720,284.076,388.658,171.783,40.985,157.828
C00689=1042.727,284.324,388.626,171.786,40.987,157.829
C00690=1042.734,284.572,388.595,171.790,40.989,157.829
C00691=1042.740,284.820,388.563,171.793,40.992,157.830
C00692=1042.747,285.068,388.532,171.797,40.994,157.831
C00693=1042.754,285.316,388.501,171.800,40.996,157.831
C00694=1042.761,285.564,388.469,171.803,40.998,157.832
C00695=1042.767,285.811,388.438,171.807,41.000,157.833
C00696=1042.774,286.059,388.406,171.811,41.003,157.833
C00697=1042.781,286.307,388.374,171.813,41.005,157.834
C00698=1042.788,286.554,388.343,171.817,41.007,157.835
C00699=1042.795,286.802,388.311,171.821,41.009,157.835
C00700=1042.801,287.050,388.280,171.824,41.012,157.836
C00701=1042.808,287.298,388.248,171.827,41.014,157.837
C00702=1042.814,287.546,388.216,171.831,41.016,157.837
C00703=1042.821,287.794,388.184,171.834,41.019,157.838
C00704=1042.828,288.042,388.152,171.837,41.021,157.839
C00705=1042.835,288.290,388.120,171.841,41.023,157.839
C00706=1042.841,288.538,388.088,171.844,41.025,157.840
C00707=1042.848,288.786,388.057,171.848,41.027,157.841
C00708=1042.855,289.033,388.025,171.851,41.029,157.841
C00709=1042.862,289.281,387.993,171.854,41.032,157.842
C00710=1042.868,289.529,387.961,171.858,41.034,157.843
C00711=1042.875,289.776,387.929,171.862,41.037,157.844
C00712=1042.882,290.025,387.897,171.866,41.039,157.844
C00713=1042.889,290.272,387.865,171.868,41.041,157.845
C00714=1042.895,290.520,387.833,171.872,41.044,157.846
C00715=1042.904,290.830,387.793,171.876,41.046,157.846
C00716=1042.912,291.141,387.753,171.881,41.050,157.847
C00717=1042.921,291.451,387.712,171.885,41.052,157.848
C00718=1042.929,291.761,387.673,171.890,41.055,157.849
C00719=1042.936,292.010,387.640,171.893,41.058,157.850
C00720=1042.942,292.258,387.609,171.897,41.060,157.851
C00721=1042.950,292.505,387.577,171.900,41.062,157.851
C00722=1042.955,292.753,387.545,171.904,41.065,157.852
C00723=1042.963,293.000,387.512,171.907,41.067,157.853
C00724=1042.970,293.248,387.480,171.911,41.070,157.853
C00725=1042.976,293.497,387.448,171.914,41.072,157.854
C00726=1042.983,293.744,387.416,171.918,41.074,157.855
C00727=1042.990,293.991,387.384,171.921,41.077,157.856
C00728=1042.997,294.240,387.351,171.925,41.079,157.856
C00729=1043.004,294.487,387.319,171.929,41.081,157.857
C00730=1043.010,294.735,387.286,171.933,41.084,157.858
C00731=1043.017,294.983,387.255,171.936,41.086,157.858
C00732=1043.024,295.231,387.222,171.939,41.089,157.859
C00733=1043.031,295.478,387.190,171.943,41.091,157.860
C00734=1043.037,295.726,387.157,171.947,41.093,157.861
C00735=1043.043,295.974,387.124,171.951,41.096,157.861
C00736=1043.051,296.222,387.092,171.953,41.098,157.862
C00737=1043.057,296.470,387.060,171.957,41.101,157.863
C00738=1043.063,296.717,387.027,171.961,41.103,157.864
C00739=1043.070,296.965,386.994,171.965,41.105,157.864
C00740=1043.077,297.213,386.962,171.969,41.108,157.865
C00741=1043.083,297.461,386.929,171.971,41.111,157.866
C00742=1043.090,297.708,386.896,171.975,41.113,157.867
C00743=1043.096,297.956,386.863,171.979,41.115,157.867
C00744=1043.103,298.204,386.830,171.983,41.118,157.868
C00745=1043.110,298.451,386.798,171.987,41.121,157.869
C00746=1043.116,298.699,386.765,171.990,41.123,157.869
C00747=1043.123,298.947,386.732,171.993,41.126,157.870
C00748=1043.129,299.195,386.700,171.997,41.128,157.871
C00749=1043.137,299.442,386.667,172.001,41.131,157.872
C00750=1043.144,299.690,386.634,172.005,41.133,157.873
C00751=1043.150,299.937,386.601,172.008,41.136,157.873
C00752=1043.156,300.185,386.568,172.012,41.138,157.874
C00753=1043.163,300.433,386.535,172.016,41.141,157.875
C00754=1043.170,300.681,386.503,172.019,41.143,157.876
C00755=1043.177,300.928,386.470,172.023,41.145,157.876
C00756=1043.183,301.176,386.437,172.027,41.148,157.877
C00757=1043.190,301.423,386.404,172.031,41.151,157.878
C00758=1043.197,301.672,386.370,172.034,41.153,157.879
C00759=1043.203,301.919,386.338,172.038,41.156,157.879
C00760=1043.210,302.167,386.306,172.041,41.158,157.880
C00761=1043.217,302.414,386.272,172.045,41.161,157.881
C00762=1043.224,302.662,386.239,172.049,41.163,157.882
C00763=1043.231,302.910,386.206,172.053,41.166,157.882
C00764=1043.237,303.158,386.173,172.057,41.169,157.883
C00765=1043.245,303.405,386.140,172.061,41.171,157.884
C00766=1043.251,303.653,386.107,172.065,41.173,157.885
C00767=1043.258,303.901,386.074,172.068,41.176,157.886
C00768=1043.265,304.148,386.041,172.071,41.179,157.886
C00769=1043.272,304.396,386.007,172.075,41.181,157.887
C00770=1043.278,304.643,385.974,172.079,41.184,157.888
C00771=1043.288,304.970,385.931,172.084,41.187,157.889
C00772=1043.296,305.297,385.887,172.089,41.191,157.890
C00773=1043.306,305.623,385.843,172.095,41.194,157.891
C00774=1043.314,305.950,385.799,172.100,41.197,157.892
C00775=1043.321,306.199,385.766,172.104,41.200,157.893
C00776=1043.329,306.446,385.733,172.107,41.202,157.894
C00777=1043.335,306.693,385.700,172.111,41.205,157.894
C00778=1043.343,306.941,385.666,172.115,41.207,157.895
C00779=1043.349,307.189,385.634,172.119,41.210,157.896
C00780=1043.356,307.436,385.600,172.123,41.213,157.897
C00781=1043.363,307.684,385.566,172.127,41.215,157.898
C00782=1043.370,307.932,385.533,172.131,41.218,157.898
C00783=1043.377,308.179,385.500,172.135,41.220,157.899
C00784=1043.384,308.427,385.467,172.139,41.223,157.900
C00785=1043.391,308.674,385.433,172.142,41.226,157.901
C00786=1043.398,308.922,385.400,172.146,41.228,157.902
C00787=1043.405,309.170,385.366,172.150,41.231,157.902
C00788=1043.412,309.417,385.333,172.154,41.233,157.903
C00789=1043.419,309.665,385.299,172.158,41.236,157.904
C00790=1043.426,309.913,385.266,172.162,41.239,157.905
C00791=1043.433,310.160,385.233,172.166,41.241,157.906
C00792=1043.440,310.408,385.199,172.170,41.244,157.906
C00793=1043.447,310.655,385.166,172.174,41.246,157.907
C00794=1043.454,310.904,385.132,172.178,41.249,157.908
C00795=1043.461,311.151,385.099,172.181,41.252,157.909
C00796=1043.468,311.398,385.065,172.185,41.254,157.910
C00797=1043.475,311.646,385.031,172.189,41.257,157.910
C00798=1043.483,311.894,384.997,172.193,41.259,157.911
C00799=1043.489,312.141,384.964,172.197,41.262,157.912
C00800=1043.496,312.389,384.931,172.201,41.265,157.913
C00801=1043.503,312.636,384.897,172.205,41.268,157.914
C00802=1043.510,312.884,384.863,172.209,41.270,157.914
C00803=1043.517,313.131,384.828,172.214,41.273,157.915
C00804=1043.524,313.378,384.795,172.218,41.276,157.916
C00805=1043.530,313.626,384.760,172.222,41.279,157.917
C00806=1043.537,313.874,384.726,172.226,41.281,157.918
C00807=1043.543,314.121,384.692,172.230,41.284,157.919
C00808=1043.551,314.369,384.659,172.234,41.287,157.920
C00809=1043.557,314.617,384.624,172.238,41.290,157.920
C00810=1043.564,314.865,384.590,172.242,41.293,157.921
C00811=1043.570,315.111,384.556,172.246,41.295,157.922
C00812=1043.578,315.359,384.522,172.250,41.299,157.923
C00813=1043.584,315.607,384.487,172.254,41.301,157.924
C00814=1043.591,315.855,384.453,172.258,41.304,157.925
C00815=1043.599,316.102,384.419,172.262,41.307,157.926
C00816=1043.605,316.349,384.385,172.265,41.310,157.926
C00817=1043.612,316.597,384.351,172.270,41.313,157.927
C00818=1043.618,316.845,384.317,172.274,41.315,157.928
C00819=1043.626,317.092,384.282,172.279,41.318,157.929
C00820=1043.632,317.340,384.248,172.282,41.321,157.930
C00821=1043.639,317.587,384.214,172.286,41.324,157.931
C00822=1043.646,317.835,384.179,172.290,41.327,157.932
C00823=1043.653,318.082,384.145,172.294,41.329,157.933
C00824=1043.660,318.329,384.110,172.298,41.333,157.934
C00825=1043.667,318.577,384.076,172.302,41.335,157.934
C00826=1043.673,318.825,384.042,172.307,41.338,157.935
C00827=1043.683,319.157,383.996,172.313,41.342,157.936
C00828=1043.692,319.488,383.950,172.318,41.346,157.938
C00829=1043.701,319.819,383.903,172.323,41.350,157.939
C00830=1043.711,320.151,383.857,172.329,41.354,157.940
C00831=1043.718,320.398,383.822,172.334,41.356,157.941
C00832=1043.725,320.646,383.788,172.338,41.360,157.942
C00833=1043.732,320.893,383.753,172.342,41.362,157.943
C00834=1043.739,321.141,383.719,172.346,41.365,157.944
C00835=1043.745,321.388,383.684,172.350,41.368,157.944
C00836=1043.753,321.635,383.649,172.355,41.371,157.945
C00837=1043.759,321.883,383.615,172.359,41.374,157.946
C00838=1043.767,322.130,383.580,172.363,41.377,157.947
C00839=1043.774,322.378,383.545,172.367,41.380,157.948
C00840=1043.781,322.625,383.511,172.371,41.383,157.949
C00841=1043.788,322.873,383.476,172.376,41.386,157.950
C00842=1043.795,323.120,383.442,172.380,41.389,157.951
C00843=1043.802,323.368,383.407,172.384,41.392,157.952
C00844=1043.809,323.616,383.372,172.388,41.395,157.953
C00845=1043.816,323.863,383.337,172.393,41.398,157.954
C00846=1043.823,324.110,383.302,172.397,41.401,157.955
C00847=1043.830,324.358,383.268,172.401,41.403,157.955
C00848=1043.837,324.605,383.233,172.405,41.406,157.956
C00849=1043.845,324.852,383.198,172.411,41.409,157.957
C00850=1043.852,325.100,383.163,172.414,41.412,157.958
C00851=1043.859,325.348,383.128,172.419,41.415,157.959
C00852=1043.866,325.595,383.093,172.424,41.418,157.960
C00853=1043.873,325.842,383.058,172.428,41.421,157.961
C00854=1043.880,326.090,383.024,172.432,41.424,157.962
C00855=1043.888,326.338,382.989,172.436,41.427,157.963
C00856=1043.895,326.585,382.954,172.441,41.430,157.964
C00857=1043.902,326.832,382.919,172.445,41.433,157.965
C00858=1043.909,327.080,382.884,172.449,41.436,157.966
C00859=1043.917,327.327,382.849,172.454,41.439,157.967
C00860=1043.924,327.575,382.814,172.458,41.442,157.968
C00861=1043.930,327.822,382.779,172.462,41.445,157.969
C00862=1043.939,328.070,382.744,172.467,41.448,157.969
C00863=1043.945,328.317,382.709,172.471,41.451,157.970
C00864=1043.953,328.564,382.674,172.476,41.455,157.971
C00865=1043.960,328.812,382.638,172.480,41.457,157.972
C00866=1043.967,329.059,382.603,172.485,41.460,157.973
C00867=1043.975,329.306,382.568,172.490,41.463,157.974
C00868=1043.982,329.554,382.533,172.494,41.466,157.975
C00869=1043.989,329.801,382.497,172.498,41.469,157.976
C00870=1043.996,330.048,382.462,172.503,41.473,157.977
C00871=1044.003,330.296,382.426,172.507,41.476,157.978
C00872=1044.010,330.544,382.391,172.511,41.479,157.979
C00873=1044.017,330.790,382.355,172.517,41.482,157.980
C00874=1044.025,331.039,382.320,172.521,41.486,157.981
C00875=1044.032,331.285,382.284,172.525,41.489,157.982
C00876=1044.038,331.533,382.249,172.530,41.492,157.983
C00877=1044.046,331.781,382.213,172.534,41.495,157.984
C00878=1044.053,332.027,382.178,172.538,41.499,157.985
C00879=1044.060,332.276,382.142,172.543,41.502,157.986
C00880=1044.067,332.523,382.106,172.548,41.505,157.987
C00881=1044.073,332.770,382.071,172.553,41.508,157.988
C00882=1044.081,333.017,382.034,172.557,41.511,157.989
C00883=1044.090,333.343,381.987,172.563,41.516,157.991
C00884=1044.100,333.671,381.940,172.569,41.520,157.992
C00885=1044.110,333.997,381.893,172.575,41.524,157.993
C00886=1044.119,334.323,381.846,172.581,41.528,157.994
C00887=1044.127,334.570,381.810,172.586,41.532,157.996
C00888=1044.133,334.818,381.775,172.590,41.535,157.997
C00889=1044.141,335.065,381.739,172.595,41.538,157.998
C00890=1044.148,335.312,381.703,172.600,41.541,157.999
C00891=1044.156,335.560,381.667,172.604,41.545,158.000
C00892=1044.162,335.807,381.631,172.609,41.548,158.001
C00893=1044.170,336.055,381.595,172.613,41.551,158.002
C00894=1044.177,336.302,381.558,172.618,41.554,158.003
C00895=1044.184,336.549,381.523,172.623,41.558,158.004
C00896=1044.191,336.797,381.486,172.628,41.561,158.005
C00897=1044.198,337.044,381.451,172.632,41.565,158.006
C00898=1044.206,337.291,381.414,172.637,41.568,158.007
C00899=1044.212,337.538,381.378,172.642,41.571,158.008
C00900=1044.220,337.786,381.342,172.647,41.574,158.009
C00901=1044.227,338.033,381.306,172.651,41.578,158.010
C00902=1044.234,338.280,381.270,172.656,41.581,158.011
C00903=1044.241,338.528,381.233,172.660,41.585,158.012
C00904=1044.248,338.774,381.197,172.666,41.588,158.013
C00905=1044.256,339.022,381.161,172.670,41.592,158.014
C00906=1044.263,339.270,381.124,172.675,41.595,158.016
C00907=1044.270,339.516,381.088,172.679,41.598,158.017
C00908=1044.278,339.764,381.052,172.685,41.602,158.018
C00909=1044.285,340.012,381.015,172.689,41.606,158.019
C00910=1044.292,340.258,380.979,172.694,41.609,158.020
C00911=1044.300,340.505,380.942,172.699,41.612,158.021
C00912=1044.307,340.753,380.906,172.704,41.616,158.022
C00913=1044.314,341.000,380.870,172.709,41.619,158.023
C00914=1044.322,341.247,380.833,172.713,41.623,158.024
C00915=1044.328,341.495,380.797,172.719,41.626,158.025
C00916=1044.336,341.742,380.760,172.723,41.629,158.026
C00917=1044.344,341.988,380.724,172.728,41.633,158.027
C00918=1044.350,342.236,380.687,172.733,41.636,158.029
C00919=1044.358,342.483,380.650,172.738,41.640,158.030
C00920=1044.365,342.731,380.613,172.743,41.644,158.031
C00921=1044.372,342.978,380.577,172.747,41.647,158.032
C00922=1044.380,343.225,380.540,172.753,41.651,158.033
C00923=1044.387,343.472,380.504,172.758,41.654,158.034
C00924=1044.395,343.719,380.466,172.762,41.658,158.035
C00925=1044.402,343.967,380.429,172.767,41.661,158.036
C00926=1044.409,344.213,380.393,172.772,41.665,158.038
C00927=1044.416,344.461,380.356,172.777,41.668,158.039
C00928=1044.424,344.708,380.319,172.782,41.672,158.040
C00929=1044.431,344.955,380.282,172.787,41.676,158.041
C00930=1044.439,345.202,380.245,172.792,41.679,158.042
C00931=1044.446,345.450,380.209,172.797,41.683,158.043
C00932=1044.453,345.697,380.171,172.802,41.686,158.044
C00933=1044.460,345.943,380.134,172.807,41.690,158.046
C00934=1044.467,346.191,380.098,172.812,41.693,158.047
C00935=1044.475,346.438,380.060,172.817,41.698,158.048
C00936=1044.482,346.685,380.023,172.822,41.701,158.049
C00937=1044.489,346.933,379.986,172.828,41.705,158.050
C00938=1044.497,347.180,379.949,172.832,41.709,158.051
C00939=1044.507,347.502,379.901,172.839,41.713,158.053
C00940=1044.517,347.825,379.851,172.846,41.718,158.055
C00941=1044.526,348.148,379.803,172.852,41.723,158.056
C00942=1044.536,348.471,379.754,172.859,41.728,158.058
C00943=1044.544,348.718,379.717,172.864,41.732,158.059
C00944=1044.551,348.965,379.679,172.869,41.735,158.060
C00945=1044.559,349.212,379.642,172.874,41.739,158.061
C00946=1044.566,349.459,379.605,172.880,41.743,158.062
C00947=1044.573,349.706,379.567,172.885,41.746,158.064
C00948=1044.581,349.953,379.531,172.889,41.750,158.065
C00949=1044.588,350.200,379.493,172.895,41.754,158.066
C00950=1044.596,350.448,379.455,172.900,41.758,158.067
C00951=1044.603,350.695,379.418,172.906,41.761,158.068
C00952=1044.610,350.942,379.380,172.910,41.766,158.070
C00953=1044.617,351.189,379.343,172.915,41.769,158.071
C00954=1044.625,351.436,379.305,172.921,41.773,158.072
C00955=1044.633,351.683,379.268,172.926,41.777,158.073
C00956=1044.640,351.929,379.230,172.932,41.781,158.075
C00957=1044.647,352.177,379.193,172.936,41.784,158.076
C00958=1044.655,352.424,379.155,172.942,41.789,158.077
C00959=1044.663,352.671,379.117,172.947,41.792,158.078
C00960=1044.670,352.918,379.079,172.953,41.796,158.079
C00961=1044.677,353.165,379.041,172.958,41.800,158.081
C00962=1044.685,353.412,379.003,172.964,41.804,158.082
C00963=1044.692,353.659,378.966,172.968,41.808,158.083
C00964=1044.700,353.907,378.928,172.974,41.812,158.085
C00965=1044.708,354.153,378.890,172.979,41.816,158.086
C00966=1044.715,354.400,378.852,172.985,41.820,158.087
C00967=1044.722,354.647,378.814,172.990,41.824,158.088
C00968=1044.730,354.894,378.776,172.995,41.827,158.089
C00969=1044.738,355.141,378.738,173.001,41.832,158.091
C00970=1044.745,355.388,378.700,173.006,41.836,158.092
C00971=1044.753,355.635,378.662,173.011,41.840,158.093
C00972=1044.760,355.883,378.624,173.016,41.843,158.095
C00973=1044.768,356.129,378.586,173.022,41.847,158.096
C00974=1044.775,356.376,378.548,173.028,41.852,158.097
C00975=1044.783,356.624,378.510,173.033,41.856,158.099
C00976=1044.791,356.870,378.471,173.039,41.860,158.100
C00977=1044.798,357.117,378.434,173.044,41.864,158.101
C00978=1044.806,357.364,378.395,173.050,41.868,158.102
C00979=1044.814,357.611,378.357,173.055,41.872,158.104
C00980=1044.821,357.857,378.319,173.061,41.876,158.105
C00981=1044.830,358.105,378.280,173.066,41.880,158.106
C00982=1044.836,358.352,378.242,173.072,41.884,158.108
C00983=1044.844,358.599,378.204,173.078,41.888,158.109
C00984=1044.852,358.846,378.165,173.083,41.892,158.110
C00985=1044.859,359.092,378.127,173.089,41.896,158.112
C00986=1044.867,359.340,378.088,173.094,41.901,158.113
C00987=1044.875,359.586,378.050,173.100,41.905,158.114
C00988=1044.882,359.833,378.011,173.105,41.909,158.116
C00989=1044.890,360.080,377.973,173.111,41.913,158.117
C00990=1044.897,360.327,377.934,173.117,41.917,158.118
C00991=1044.906,360.574,377.896,173.122,41.921,158.120
C00992=1044.913,360.820,377.858,173.128,41.926,158.121
C00993=1044.921,361.068,377.818,173.133,41.930,158.122
C00994=1044.928,361.314,377.780,173.139,41.934,158.124
C00995=1044.938,361.643,377.728,173.146,41.939,158.126
C00996=1044.949,361.971,377.677,173.153,41.946,158.128
C00997=1044.960,362.300,377.625,173.162,41.951,158.129
C00998=1044.970,362.629,377.574,173.169,41.957,158.131
C00999=1044.977,362.875,377.535,173.174,41.961,158.133
C01000=1044.985,363.122,377.495,173.180,41.965,158.134
C01001=1044.993,363.369,377.457,173.186,41.970,158.135
C01002=1045.000,363.616,377.418,173.192,41.974,158.137
C01003=1045.008,363.863,377.379,173.198,41.978,158.138
C01004=1045.015,364.109,377.340,173.204,41.983,158.140
C01005=1045.024,364.356,377.300,173.210,41.987,158.141
C01006=1045.031,364.603,377.262,173.215,41.991,158.142
C01007=1045.039,364.849,377.222,173.221,41.996,158.144
C01008=1045.046,365.097,377.183,173.227,42.000,158.145
C01009=1045.054,365.343,377.144,173.232,42.005,158.147
C01010=1045.062,365.590,377.104,173.238,42.009,158.148
C01011=1045.070,365.837,377.066,173.245,42.014,158.150
C01012=1045.077,366.083,377.026,173.250,42.018,158.151
C01013=1045.085,366.330,376.987,173.256,42.022,158.153
C01014=1045.093,366.577,376.947,173.262,42.027,158.154
C01015=1045.101,366.824,376.908,173.268,42.032,158.156
C01016=1045.109,367.070,376.869,173.273,42.036,158.157
C01017=1045.116,367.318,376.829,173.280,42.040,158.158
C01018=1045.125,367.564,376.790,173.286,42.045,158.160
C01019=1045.132,367.811,376.750,173.292,42.049,158.161
C01020=1045.140,368.057,376.711,173.298,42.054,158.163
C01021=1045.148,368.304,376.671,173.303,42.059,158.164
C01022=1045.156,368.550,376.632,173.310,42.063,158.166
C01023=1045.164,368.798,376.593,173.316,42.068,158.167
C01024=1045.172,369.045,376.553,173.322,42.072,158.169
C01025=1045.180,369.292,376.514,173.327,42.077,158.170
C01026=1045.188,369.538,376.474,173.334,42.081,158.172
C01027=1045.196,369.784,376.435,173.340,42.086,158.173
C01028=1045.203,370.031,376.395,173.346,42.091,158.175
C01029=1045.212,370.278,376.355,173.353,42.095,158.176
C01030=1045.220,370.524,376.315,173.358,42.100,158.178
C01031=1045.228,370.771,376.275,173.364,42.104,158.179
C01032=1045.236,371.018,376.236,173.371,42.109,158.181
C01033=1045.244,371.265,376.196,173.377,42.114,158.183
C01034=1045.251,371.511,376.156,173.383,42.118,158.184
C01035=1045.259,371.758,376.115,173.389,42.123,158.186
C01036=1045.268,372.004,376.076,173.396,42.128,158.187
C01037=1045.276,372.251,376.036,173.401,42.133,158.189
C01038=1045.284,372.497,375.995,173.407,42.137,158.190
C01039=1045.291,372.744,375.955,173.414,42.142,158.192
C01040=1045.299,372.991,375.915,173.420,42.147,158.193
C01041=1045.307,373.238,375.875,173.426,42.152,158.195
C01042=1045.315,373.484,375.835,173.433,42.156,158.197
C01043=1045.323,373.731,375.794,173.439,42.162,158.198
C01044=1045.331,373.977,375.755,173.446,42.166,158.200
C01045=1045.339,374.224,375.714,173.452,42.171,158.201
C01046=1045.347,374.471,375.674,173.458,42.176,158.203
C01047=1045.355,374.717,375.634,173.465,42.181,158.205
C01048=1045.363,374.963,375.593,173.471,42.186,158.206
C01049=1045.371,375.210,375.553,173.477,42.190,158.208
C01050=1045.379,375.456,375.512,173.483,42.195,158.209
C01051=1045.391,375.805,375.455,173.492,42.203,158.212
C01052=1045.402,376.152,375.398,173.502,42.209,158.214
C01053=1045.414,376.501,375.341,173.511,42.216,158.216
C01054=1045.425,376.848,375.284,173.520,42.223,158.219
C01055=1045.434,377.095,375.243,173.527,42.228,158.220
C01056=1045.442,377.341,375.203,173.533,42.233,158.222
C01057=1045.450,377.588,375.162,173.540,42.238,158.224
C01058=1045.458,377.834,375.121,173.546,42.243,158.225
C01059=1045.466,378.081,375.080,173.553,42.248,158.227
C01060=1045.474,378.327,375.040,173.559,42.253,158.229
C01061=1045.482,378.574,374.999,173.566,42.258,158.230
C01062=1045.491,378.821,374.958,173.572,42.263,158.232
C01063=1045.499,379.067,374.918,173.579,42.269,158.234
C01064=1045.507,379.313,374.877,173.585,42.274,158.235
C01065=1045.516,379.560,374.836,173.592,42.279,158.237
C01066=1045.524,379.806,374.795,173.599,42.284,158.239
C01067=1045.531,380.052,374.753,173.605,42.289,158.240
C01068=1045.540,380.299,374.712,173.612,42.294,158.242
C01069=1045.548,380.546,374.672,173.618,42.299,158.244
C01070=1045.556,380.791,374.630,173.625,42.304,158.246
C01071=1045.564,381.039,374.589,173.632,42.310,158.247
C01072=1045.572,381.285,374.548,173.639,42.315,158.249
C01073=1045.581,381.531,374.506,173.646,42.320,158.251
C01074=1045.589,381.778,374.466,173.652,42.326,158.253
C01075=1045.597,382.024,374.424,173.659,42.331,158.254
C01076=1045.605,382.271,374.383,173.666,42.336,158.256
C01077=1045.614,382.516,374.341,173.672,42.341,158.258
C01078=1045.622,382.763,374.300,173.680,42.347,158.260
C01079=1045.630,383.009,374.259,173.687,42.352,158.262
C01080=1045.639,383.256,374.218,173.693,42.357,158.263
C01081=1045.647,383.502,374.176,173.700,42.363,158.265
C01082=1045.655,383.748,374.134,173.707,42.368,158.267
C01083=1045.663,383.995,374.093,173.714,42.373,158.269
C01084=1045.672,384.241,374.052,173.721,42.379,158.271
C01085=1045.681,384.487,374.010,173.728,42.384,158.272
C01086=1045.689,384.733,373.968,173.735,42.389,158.274
C01087=1045.698,384.980,373.926,173.741,42.395,158.276
C01088=1045.706,385.226,373.885,173.749,42.400,158.278
C01089=1045.714,385.473,373.843,173.756,42.406,158.280
C01090=1045.723,385.719,373.801,173.763,42.411,158.282
C01091=1045.732,385.965,373.760,173.770,42.417,158.283
C01092=1045.739,386.211,373.718,173.777,42.423,158.285
C01093=1045.748,386.458,373.676,173.784,42.428,158.287
C01094=1045.757,386.704,373.634,173.791,42.434,158.289
C01095=1045.765,386.950,373.592,173.799,42.439,158.291
C01096=1045.774,387.197,373.551,173.806,42.444,158.293
C01097=1045.783,387.443,373.509,173.812,42.450,158.295
C01098=1045.791,387.690,373.467,173.820,42.456,158.297
C01099=1045.800,387.935,373.424,173.827,42.461,158.298
C01100=1045.808,388.181,373.383,173.834,42.467,158.300
C01101=1045.816,388.428,373.341,173.841,42.472,158.302
C01102=1045.825,388.674,373.299,173.849,42.478,158.304
C01103=1045.834,388.920,373.256,173.856,42.483,158.306
C01104=1045.843,389.166,373.214,173.864,42.489,158.308
C01105=1045.851,389.413,373.172,173.870,42.495,158.310
C01106=1045.860,389.658,373.130,173.877,42.501,158.312
C01107=1045.873,390.040,373.064,173.889,42.510,158.315
C01108=1045.886,390.421,372.999,173.901,42.518,158.318
C01109=1045.900,390.803,372.933,173.912,42.528,158.321
C01110=1045.913,391.184,372.867,173.924,42.537,158.324
C01111=1045.922,391.430,372.824,173.931,42.543,158.326
C01112=1045.930,391.676,372.781,173.938,42.548,158.328
C01113=1045.939,391.922,372.739,173.946,42.554,158.330
C01114=1045.948,392.168,372.697,173.953,42.560,158.332
C01115=1045.956,392.414,372.654,173.961,42.566,158.334
C01116=1045.965,392.660,372.611,173.968,42.572,158.336
C01117=1045.973,392.906,372.568,173.976,42.577,158.338
C01118=1045.982,393.153,372.526,173.983,42.583,158.340
C01119=1045.991,393.399,372.483,173.991,42.589,158.342
C01120=1046.000,393.645,372.439,173.998,42.595,158.344
C01121=1046.008,393.891,372.396,174.006,42.601,158.346
C01122=1046.018,394.137,372.354,174.015,42.608,158.348
C01123=1046.026,394.383,372.311,174.022,42.614,158.350
C01124=1046.035,394.629,372.267,174.030,42.620,158.353
C01125=1046.043,394.875,372.224,174.037,42.626,158.355
C01126=1046.052,395.121,372.181,174.045,42.632,158.357
C01127=1046.062,395.367,372.138,174.052,42.638,158.359
C01128=1046.070,395.613,372.095,174.060,42.644,158.361
C01129=1046.079,395.859,372.052,174.069,42.650,158.363
C01130=1046.088,396.105,372.008,174.076,42.656,158.365
C01131=1046.097,396.352,371.965,174.084,42.662,158.367
C01132=1046.105,396.598,371.922,174.092,42.668,158.369
C01133=1046.114,396.843,371.878,174.099,42.675,158.372
C01134=1046.123,397.090,371.835,174.108,42.681,158.374
C01135=1046.132,397.335,371.791,174.116,42.687,158.376
C01136=1046.140,397.581,371.748,174.124,42.694,158.378
C01137=1046.150,397.827,371.704,174.131,42.700,158.380
C01138=1046.158,398.073,371.661,174.139,42.706,158.382
C01139=1046.167,398.319,371.617,174.148,42.713,158.385
C01140=1046.176,398.565,371.573,174.155,42.718,158.387
C01141=1046.185,398.811,371.530,174.163,42.725,158.389
C01142=1046.194,399.057,371.486,174.172,42.731,158.391
C01143=1046.203,399.303,371.442,174.180,42.738,158.393
C01144=1046.213,399.549,371.398,174.187,42.744,158.396
C01145=1046.221,399.795,371.355,174.196,42.751,158.398
C01146=1046.230,400.041,371.311,174.204,42.757,158.400
C01147=1046.239,400.286,371.267,174.212,42.764,158.402
C01148=1046.249,400.533,371.223,174.221,42.770,158.405
C01149=1046.258,400.778,371.180,174.229,42.776,158.407
C01150=1046.267,401.024,371.135,174.237,42.783,158.409
C01151=1046.276,401.270,371.091,174.245,42.789,158.411
C01152=1046.285,401.516,371.048,174.253,42.796,158.414
C01153=1046.295,401.762,371.003,174.262,42.803,158.416
C01154=1046.303,402.008,370.959,174.270,42.809,158.418
C01155=1046.312,402.254,370.915,174.279,42.816,158.421
C01156=1046.321,402.500,370.871,174.287,42.822,158.423
C01157=1046.331,402.745,370.826,174.296,42.829,158.425
C01158=1046.340,402.991,370.782,174.304,42.836,158.428
C01159=1046.349,403.237,370.738,174.313,42.842,158.430
C01160=1046.358,403.483,370.693,174.320,42.849,158.432
C01161=1046.367,403.728,370.649,174.329,42.856,158.435
C01162=1046.376,403.975,370.604,174.337,42.862,158.437
C01163=1046.392,404.375,370.531,174.351,42.874,158.441
C01164=1046.406,404.775,370.459,174.365,42.884,158.445
C01165=1046.421,405.175,370.385,174.379,42.896,158.449
C01166=1046.437,405.576,370.313,174.393,42.907,158.453
C01167=1046.445,405.821,370.268,174.402,42.914,158.455
C01168=1046.455,406.067,370.223,174.411,42.921,158.458
C01169=1046.464,406.313,370.178,174.419,42.928,158.460
C01170=1046.473,406.559,370.134,174.428,42.935,158.462
C01171=1046.482,406.805,370.088,174.438,42.941,158.465
C01172=1046.492,407.050,370.044,174.446,42.949,158.467
C01173=1046.501,407.296,369.998,174.455,42.956,158.470
C01174=1046.510,407.541,369.953,174.464,42.962,158.472
C01175=1046.520,407.787,369.909,174.472,42.970,158.475
C01176=1046.530,408.033,369.863,174.481,42.977,158.477
C01177=1046.539,408.279,369.818,174.491,42.984,158.480
C01178=1046.548,408.525,369.773,174.500,42.991,158.482
C01179=1046.558,408.770,369.728,174.508,42.998,158.485
C01180=1046.567,409.016,369.682,174.517,43.005,158.487
C01181=1046.577,409.261,369.637,174.527,43.012,158.490
C01182=1046.586,409.507,369.591,174.536,43.019,158.493
C01183=1046.596,409.753,369.546,174.545,43.027,158.495
C01184=1046.605,409.999,369.501,174.554,43.034,158.498
C01185=1046.615,410.244,369.455,174.563,43.041,158.500
C01186=1046.625,410.490,369.409,174.572,43.049,158.503
C01187=1046.634,410.735,369.363,174.581,43.056,158.506
C01188=1046.644,410.981,369.318,174.591,43.063,158.508
C01189=1046.654,411.227,369.272,174.600,43.070,158.511
C01190=1046.664,411.472,369.227,174.609,43.077,158.513
C01191=1046.673,411.718,369.181,174.619,43.085,158.516
C01192=1046.683,411.964,369.136,174.628,43.092,158.519
C01193=1046.692,412.209,369.090,174.638,43.100,158.521
C01194=1046.703,412.455,369.044,174.647,43.107,158.524
C01195=1046.712,412.700,368.998,174.656,43.114,158.527
C01196=1046.722,412.946,368.952,174.666,43.122,158.529
C01197=1046.731,413.192,368.906,174.675,43.129,158.532
C01198=1046.741,413.437,368.859,174.685,43.137,158.535
C01199=1046.751,413.682,368.814,174.694,43.144,158.538
C01200=1046.761,413.928,368.767,174.704,43.152,158.540
C01201=1046.770,414.173,368.721,174.713,43.160,158.543
C01202=1046.780,414.419,368.674,174.724,43.167,158.546
C01203=1046.789,414.665,368.628,174.733,43.175,158.549
C01204=1046.799,414.910,368.582,174.743,43.183,158.551
C01205=1046.809,415.156,368.536,174.753,43.191,158.554
C01206=1046.820,415.401,368.489,174.762,43.198,158.557
C01207=1046.829,415.647,368.443,174.772,43.206,158.560
C01208=1046.839,415.892,368.396,174.782,43.214,158.563
C01209=1046.849,416.137,368.349,174.792,43.222,158.566
C01210=1046.859,416.383,368.303,174.802,43.229,158.568
C01211=1046.869,416.629,368.256,174.811,43.237,158.571
C01212=1046.878,416.873,368.209,174.822,43.245,158.574
C01213=1046.888,417.119,368.163,174.832,43.252,158.577
C01214=1046.898,417.365,368.116,174.841,43.261,158.580
C01215=1046.909,417.610,368.070,174.852,43.268,158.583
C01216=1046.919,417.855,368.023,174.862,43.276,158.586
C01217=1046.929,418.101,367.975,174.872,43.284,158.589
C01218=1046.939,418.347,367.929,174.882,43.292,158.591
C01219=1046.955,418.724,367.856,174.898,43.304,158.596
C01220=1046.970,419.102,367.784,174.914,43.317,158.601
C01221=1046.986,419.480,367.711,174.930,43.330,158.605
C01222=1047.001,419.857,367.638,174.945,43.342,158.610
C01223=1047.011,420.103,367.590,174.956,43.350,158.613
C01224=1047.021,420.348,367.543,174.967,43.358,158.616
C01225=1047.031,420.594,367.496,174.977,43.367,158.619
C01226=1047.042,420.838,367.448,174.988,43.375,158.622
C01227=1047.052,421.084,367.401,174.998,43.383,158.625
C01228=1047.062,421.329,367.354,175.009,43.391,158.628
C01229=1047.072,421.575,367.305,175.019,43.400,158.631
C01230=1047.083,421.820,367.258,175.030,43.408,158.634
C01231=1047.094,422.095,367.204,175.041,43.418,158.638
C01232=1047.105,422.370,367.151,175.054,43.426,158.641
C01233=1047.118,422.645,367.097,175.066,43.436,158.645
C01234=1047.129,422.920,367.044,175.078,43.446,158.648
C01235=1047.139,423.165,366.995,175.089,43.454,158.651
C01236=1047.150,423.411,366.948,175.100,43.462,158.655
C01237=1047.160,423.655,366.900,175.110,43.471,158.658
C01238=1047.171,423.900,366.852,175.122,43.480,158.661
C01239=1047.181,424.146,366.804,175.133,43.488,158.664
C01240=1047.191,424.391,366.756,175.144,43.497,158.668
C01241=1047.202,424.636,366.708,175.155,43.505,158.671
C01242=1047.213,424.881,366.660,175.166,43.514,158.674
C01243=1047.224,425.126,366.611,175.177,43.522,158.677
C01244=1047.234,425.371,366.563,175.188,43.531,158.680
C01245=1047.245,425.617,366.514,175.199,43.540,158.684
C01246=1047.254,425.862,366.466,175.211,43.549,158.687
C01247=1047.266,426.107,366.418,175.222,43.557,158.690
C01248=1047.276,426.351,366.368,175.233,43.566,158.694
C01249=1047.287,426.597,366.320,175.244,43.575,158.697
C01250=1047.297,426.841,366.272,175.256,43.584,158.700
C01251=1047.308,427.086,366.223,175.267,43.593,158.704
C01252=1047.319,427.332,366.174,175.279,43.602,158.707
C01253=1047.329,427.576,366.125,175.290,43.610,158.710
C01254=1047.340,427.821,366.077,175.303,43.619,158.714
C01255=1047.351,428.066,366.027,175.314,43.628,158.717
C01256=1047.361,428.311,365.979,175.326,43.637,158.721
C01257=1047.372,428.556,365.930,175.337,43.646,158.724
C01258=1047.383,428.801,365.881,175.349,43.656,158.728
C01259=1047.394,429.047,365.832,175.360,43.665,158.731
C01260=1047.405,429.291,365.783,175.373,43.673,158.735
C01261=1047.415,429.536,365.733,175.385,43.683,158.738
C01262=1047.426,429.781,365.684,175.396,43.692,158.742
C01263=1047.437,430.025,365.635,175.409,43.701,158.745
C01264=1047.448,430.271,365.585,175.420,43.710,158.749
C01265=1047.459,430.516,365.536,175.432,43.720,158.752
C01266=1047.469,430.761,365.486,175.445,43.729,158.756
C01267=1047.481,431.005,365.436,175.457,43.738,158.760
C01268=1047.492,431.250,365.387,175.468,43.748,158.763
C01269=1047.502,431.495,365.337,175.481,43.757,158.767
C01270=1047.514,431.740,365.288,175.493,43.766,158.770
C01271=1047.525,431.984,365.238,175.506,43.776,158.774
C01272=1047.535,432.229,365.188,175.518,43.786,158.778
C01273=1047.546,432.474,365.138,175.531,43.795,158.782
C01274=1047.558,432.718,365.089,175.542,43.804,158.785
C01275=1047.568,432.934,365.044,175.554,43.813,158.788
C01276=1047.578,433.149,365.000,175.565,43.821,158.792
C01277=1047.587,433.365,364.957,175.575,43.830,158.795
C01278=1047.597,433.580,364.912,175.587,43.838,158.798
C01279=1047.607,433.795,364.868,175.598,43.846,158.802
C01280=1047.617,434.010,364.824,175.610,43.855,158.805
C01281=1047.627,434.226,364.780,175.620,43.864,158.808
C01282=1047.636,434.441,364.735,175.632,43.872,158.812
C01283=1047.648,434.686,364.685,175.645,43.882,158.816
C01284=1047.660,434.930,364.635,175.658,43.891,158.819
C01285=1047.671,435.175,364.584,175.671,43.901,158.823
C01286=1047.682,435.420,364.534,175.683,43.911,158.827
C01287=1047.694,435.665,364.483,175.696,43.921,158.831
C01288=1047.706,435.909,364.433,175.709,43.931,158.835
C01289=1047.717,436.154,364.383,175.723,43.941,158.839
C01290=1047.728,436.398,364.332,175.736,43.951,158.843
C01291=1047.740,436.643,364.281,175.749,43.961,158.847
C01292=1047.751,436.888,364.231,175.762,43.970,158.851
C01293=1047.763,437.132,364.179,175.776,43.981,158.855
C01294=1047.774,437.376,364.128,175.789,43.991,158.859
C01295=1047.786,437.621,364.078,175.802,44.001,158.863
C01296=1047.798,437.866,364.026,175.816,44.011,158.867
C01297=1047.809,438.109,363.975,175.829,44.021,158.871
C01298=1047.820,438.355,363.924,175.843,44.032,158.875
C01299=1047.832,438.599,363.873,175.856,44.042,158.879
C01300=1047.844,438.844,363.822,175.870,44.052,158.883
C01301=1047.856,439.087,363.771,175.884,44.062,158.887
C01302=1047.867,439.332,363.719,175.898,44.073,158.891
C01303=1047.879,439.576,363.668,175.911,44.083,158.895
C01304=1047.891,439.821,363.616,175.926,44.093,158.900
C01305=1047.903,440.065,363.564,175.939,44.103,158.904
C01306=1047.914,440.310,363.512,175.953,44.114,158.908
C01307=1047.926,440.554,363.461,175.968,44.124,158.912
C01308=1047.939,440.798,363.409,175.981,44.135,158.917
C01309=1047.950,441.043,363.357,175.995,44.146,158.921
C01310=1047.962,441.287,363.306,176.010,44.156,158.925
C01311=1047.975,441.531,363.254,176.024,44.167,158.929
C01312=1047.987,441.775,363.202,176.039,44.178,158.934
C01313=1047.998,442.020,363.150,176.052,44.188,158.938
C01314=1048.010,442.264,363.098,176.067,44.199,158.942
C01315=1048.022,442.507,363.045,176.082,44.209,158.947
C01316=1048.034,442.751,362.993,176.096,44.221,158.951
C01317=1048.046,442.996,362.941,176.111,44.231,158.956
C01318=1048.059,443.240,362.888,176.126,44.242,158.960
C01319=1048.071,443.484,362.836,176.140,44.253,158.965
C01320=1048.083,443.728,362.784,176.155,44.264,158.969
C01321=1048.095,443.973,362.731,176.170,44.275,158.974
C01322=1048.107,444.217,362.679,176.185,44.285,158.978
C01323=1048.119,444.461,362.627,176.199,44.297,158.982
C01324=1048.133,444.705,362.573,176.214,44.308,158.987
C01325=1048.144,444.949,362.521,176.230,44.319,158.992
C01326=1048.157,445.193,362.468,176.245,44.330,158.996
C01327=1048.169,445.436,362.416,176.260,44.341,159.001
C01328=1048.181,445.679,362.363,176.275,44.352,159.006
C01329=1048.194,445.922,362.311,176.290,44.363,159.010
C01330=1048.208,446.166,362.259,176.306,44.374,159.015
C01331=1048.222,446.409,362.207,176.322,44.385,159.019
C01332=1048.237,446.653,362.156,176.337,44.395,159.024
C01333=1048.253,446.897,362.106,176.353,44.406,159.028
C01334=1048.269,447.141,362.056,176.368,44.416,159.033
C01335=1048.298,447.545,361.974,176.395,44.433,159.040
C01336=1048.328,447.949,361.894,176.421,44.450,159.047
C01337=1048.360,448.354,361.816,176.447,44.466,159.055
C01338=1048.394,448.760,361.738,176.475,44.481,159.062
C01339=1048.415,449.005,361.692,176.491,44.491,159.066
C01340=1048.437,449.250,361.647,176.507,44.500,159.070
C01341=1048.460,449.494,361.602,176.524,44.509,159.075
C01342=1048.484,449.739,361.558,176.540,44.518,159.079
C01343=1048.507,449.984,361.514,176.557,44.527,159.083
C01344=1048.532,450.231,361.471,176.573,44.535,159.087
C01345=1048.558,450.475,361.428,176.590,44.544,159.091
C01346=1048.584,450.721,361.386,176.607,44.552,159.095
C01347=1048.274,450.752,361.082,176.608,44.641,159.121
C01348=1048.248,450.507,361.124,176.591,44.633,159.117
C01349=1048.222,450.261,361.167,176.574,44.624,159.113
C01350=1048.197,450.016,361.210,176.557,44.616,159.109
C01351=1048.172,449.770,361.254,176.540,44.607,159.105
C01352=1048.149,449.526,361.298,176.524,44.598,159.100
C01353=1048.126,449.280,361.343,176.507,44.590,159.096
C01354=1048.104,449.036,361.388,176.491,44.580,159.092
C01355=1048.082,448.791,361.434,176.475,44.571,159.088
C01356=1048.049,448.403,361.508,176.449,44.556,159.081
C01357=1048.018,448.015,361.583,176.423,44.541,159.074
C01358=1047.989,447.628,361.659,176.398,44.525,159.067
C01359=1047.961,447.242,361.737,176.373,44.509,159.060
C01360=1047.944,446.998,361.786,176.357,44.500,159.056
C01361=1047.927,446.754,361.837,176.341,44.489,159.051
C01362=1047.912,446.510,361.887,176.325,44.478,159.047
C01363=1047.898,446.267,361.938,176.310,44.468,159.042
C01364=1047.885,446.023,361.989,176.294,44.457,159.038
C01365=1047.871,445.779,362.042,176.279,44.446,159.033
C01366=1047.859,445.537,362.095,176.263,44.435,159.028
C01367=1047.846,445.294,362.147,176.248,44.424,159.024
C01368=1047.834,445.050,362.200,176.233,44.413,159.019
C01369=1047.821,444.806,362.253,176.218,44.402,159.014
C01370=1047.809,444.562,362.305,176.203,44.391,159.010
C01371=1047.796,444.318,362.358,176.187,44.380,159.005
C01372=1047.784,444.074,362.411,176.172,44.369,159.001
C01373=1047.772,443.829,362.463,176.158,44.358,158.996
C01374=1047.759,443.585,362.515,176.143,44.347,158.992
C01375=1047.747,443.341,362.567,176.128,44.336,158.987
C01376=1047.735,443.096,362.621,176.113,44.326,158.983
C01377=1047.723,442.853,362.673,176.099,44.315,158.978
C01378=1047.711,442.609,362.725,176.084,44.304,158.974
C01379=1047.699,442.365,362.777,176.069,44.294,158.970
C01380=1047.687,442.121,362.830,176.055,44.283,158.965
C01381=1047.674,441.876,362.882,176.040,44.272,158.961
C01382=1047.662,441.632,362.934,176.025,44.262,158.957
C01383=1047.650,441.388,362.986,176.012,44.251,158.952
C01384=1047.638,441.144,363.038,175.997,44.241,158.948
C01385=1047.626,440.899,363.089,175.983,44.230,158.944
C01386=1047.614,440.655,363.141,175.968,44.220,158.939
C01387=1047.603,440.410,363.193,175.955,44.209,158.935
C01388=1047.591,440.166,363.245,175.941,44.199,158.931
C01389=1047.579,439.922,363.297,175.926,44.189,158.927
C01390=1047.567,439.678,363.348,175.913,44.178,158.922
C01391=1047.556,439.434,363.399,175.899,44.168,158.918
C01392=1047.544,439.189,363.451,175.884,44.158,158.914
C01393=1047.532,438.945,363.502,175.871,44.147,158.910
C01394=1047.520,438.700,363.553,175.857,44.137,158.906
C01395=1047.508,438.456,363.605,175.844,44.127,158.902
C01396=1047.497,438.212,363.656,175.829,44.117,158.898
C01397=1047.485,437.967,363.707,175.816,44.107,158.894
C01398=1047.473,437.722,363.758,175.802,44.097,158.890
C01399=1047.461,437.478,363.809,175.789,44.087,158.885
C01400=1047.450,437.234,363.860,175.776,44.076,158.881
C01401=1047.439,436.989,363.911,175.762,44.067,158.878
C01402=1047.427,436.745,363.962,175.749,44.057,158.873
C01403=1047.416,436.500,364.013,175.736,44.047,158.870
C01404=1047.404,436.255,364.064,175.722,44.037,158.866
C01405=1047.393,436.011,364.115,175.709,44.027,158.862
C01406=1047.381,435.766,364.165,175.696,44.017,158.858
C01407=1047.370,435.522,364.215,175.683,44.008,158.854
C01408=1047.358,435.277,364.266,175.670,43.998,158.850
C01409=1047.347,435.033,364.317,175.657,43.988,158.846
C01410=1047.335,434.788,364.367,175.644,43.978,158.842
C01411=1047.323,434.544,364.417,175.631,43.969,158.838
C01412=1047.314,434.327,364.462,175.620,43.960,158.835
C01413=1047.303,434.110,364.506,175.608,43.951,158.832
C01414=1047.293,433.894,364.550,175.597,43.943,158.828
C01415=1047.284,433.678,364.595,175.585,43.935,158.825
C01416=1047.274,433.462,364.639,175.575,43.926,158.822
C01417=1047.264,433.245,364.683,175.564,43.918,158.818
C01418=1047.254,433.028,364.728,175.552,43.910,158.815
C01419=1047.244,432.812,364.772,175.541,43.901,158.812
C01420=1047.233,432.567,364.822,175.529,43.891,158.808
C01421=1047.222,432.323,364.871,175.516,43.882,158.804
C01422=1047.211,432.078,364.921,175.504,43.873,158.801
C01423=1047.200,431.834,364.971,175.491,43.863,158.797
C01424=1047.189,431.589,365.020,175.479,43.854,158.793
C01425=1047.178,431.344,365.071,175.466,43.845,158.790
C01426=1047.167,431.099,365.120,175.455,43.835,158.786
C01427=1047.156,430.854,365.170,175.442,43.826,158.783
C01428=1047.145,430.610,365.219,175.430,43.817,158.779
C01429=1047.134,430.365,365.269,175.417,43.808,158.775
C01430=1047.123,430.120,365.319,175.406,43.799,158.772
C01431=1047.112,429.875,365.368,175.394,43.789,158.768
C01432=1047.101,429.630,365.417,175.381,43.780,158.765
C01433=1047.090,429.385,365.467,175.370,43.771,158.761
C01434=1047.079,429.140,365.516,175.358,43.762,158.758
C01435=1047.069,428.895,365.565,175.347,43.753,158.754
C01436=1047.059,428.650,365.614,175.334,43.744,158.751
C01437=1047.047,428.406,365.663,175.322,43.735,158.747
C01438=1047.036,428.161,365.712,175.311,43.726,158.744
C01439=1047.025,427.915,365.761,175.299,43.717,158.740
C01440=1047.015,427.671,365.810,175.288,43.708,158.737
C01441=1047.004,427.426,365.859,175.275,43.699,158.733
C01442=1046.993,427.181,365.908,175.264,43.690,158.730
C01443=1046.982,426.935,365.957,175.253,43.682,158.727
C01444=1046.972,426.691,366.005,175.241,43.673,158.723
C01445=1046.961,426.445,366.054,175.230,43.664,158.720
C01446=1046.951,426.201,366.102,175.218,43.655,158.717
C01447=1046.940,425.955,366.150,175.207,43.647,158.713
C01448=1046.930,425.711,366.200,175.195,43.638,158.710
C01449=1046.919,425.466,366.248,175.184,43.629,158.707
C01450=1046.909,425.221,366.296,175.173,43.621,158.703
C01451=1046.898,424.975,366.345,175.162,43.612,158.700
C01452=1046.887,424.731,366.393,175.150,43.604,158.697
C01453=1046.877,424.485,366.442,175.139,43.595,158.694
C01454=1046.866,424.240,366.490,175.128,43.587,158.690
C01455=1046.856,423.994,366.537,175.118,43.578,158.687
C01456=1046.845,423.750,366.585,175.106,43.569,158.684
C01457=1046.835,423.504,366.634,175.095,43.561,158.681
C01458=1046.824,423.259,366.682,175.084,43.553,158.678
C01459=1046.814,423.014,366.729,175.073,43.544,158.674
C01460=1046.803,422.769,366.777,175.063,43.536,158.671
C01461=1046.793,422.523,366.825,175.052,43.527,158.668
C01462=1046.782,422.279,366.872,175.041,43.519,158.665
C01463=1046.772,422.033,366.921,175.030,43.511,158.662
C01464=1046.762,421.788,366.969,175.020,43.503,158.659
C01465=1046.751,421.543,367.016,175.008,43.494,158.656
C01466=1046.741,421.298,367.064,174.997,43.486,158.653
C01467=1046.731,421.053,367.111,174.988,43.478,158.649
C01468=1046.721,420.807,367.159,174.977,43.470,158.646
C01469=1046.711,420.562,367.206,174.967,43.461,158.643
C01470=1046.700,420.316,367.254,174.956,43.453,158.640
C01471=1046.690,420.071,367.301,174.946,43.445,158.637
C01472=1046.673,419.662,367.381,174.928,43.432,158.632
C01473=1046.657,419.252,367.459,174.911,43.418,158.627
C01474=1046.640,418.843,367.538,174.893,43.405,158.622
C01475=1046.623,418.433,367.617,174.876,43.391,158.617
C01476=1046.612,418.187,367.664,174.866,43.384,158.614
C01477=1046.602,417.941,367.710,174.855,43.376,158.611
C01478=1046.592,417.696,367.757,174.845,43.368,158.609
C01479=1046.582,417.451,367.805,174.836,43.360,158.606
C01480=1046.572,417.205,367.851,174.825,43.352,158.603
C01481=1046.563,416.960,367.898,174.815,43.344,158.600
C01482=1046.553,416.715,367.945,174.806,43.336,158.597
C01483=1046.543,416.469,367.992,174.795,43.329,158.594
C01484=1046.532,416.224,368.038,174.785,43.321,158.591
C01485=1046.522,415.978,368.085,174.776,43.313,158.589
C01486=1046.512,415.733,368.131,174.765,43.306,158.586
C01487=1046.503,415.487,368.178,174.755,43.298,158.583
C01488=1046.493,415.241,368.224,174.746,43.290,158.580
C01489=1046.483,414.997,368.271,174.736,43.282,158.577
C01490=1046.473,414.751,368.317,174.726,43.275,158.574
C01491=1046.463,414.505,368.363,174.716,43.268,158.572
C01492=1046.447,414.099,368.441,174.700,43.255,158.567
C01493=1046.431,413.691,368.517,174.684,43.242,158.562
C01494=1046.415,413.284,368.593,174.668,43.230,158.558
C01495=1046.399,412.878,368.670,174.652,43.218,158.553
C01496=1046.389,412.631,368.716,174.643,43.210,158.551
C01497=1046.380,412.386,368.762,174.633,43.202,158.548
C01498=1046.369,412.141,368.808,174.624,43.195,158.545
C01499=1046.360,411.894,368.854,174.615,43.188,158.543
C01500=1046.350,411.649,368.900,174.605,43.181,158.540
C01501=1046.340,411.404,368.945,174.596,43.173,158.537
C01502=1046.331,411.157,368.991,174.586,43.166,158.535
C01503=1046.321,410.913,369.037,174.577,43.159,158.532
C01504=1046.311,410.666,369.082,174.568,43.151,158.530
C01505=1046.301,410.421,369.128,174.558,43.144,158.527
C01506=1046.292,410.175,369.173,174.549,43.137,158.524
C01507=1046.282,409.930,369.218,174.540,43.130,158.522
C01508=1046.273,409.684,369.265,174.530,43.123,158.519
C01509=1046.263,409.438,369.310,174.521,43.116,158.517
C01510=1046.254,409.193,369.355,174.513,43.109,158.514
C01511=1046.244,408.947,369.400,174.504,43.101,158.511
C01512=1046.234,408.701,369.446,174.494,43.095,158.509
C01513=1046.225,408.456,369.491,174.485,43.087,158.506
C01514=1046.216,408.210,369.537,174.476,43.080,158.504
C01515=1046.206,407.964,369.581,174.467,43.074,158.501
C01516=1046.197,407.719,369.627,174.458,43.066,158.499
C01517=1046.187,407.473,369.672,174.449,43.059,158.496
C01518=1046.178,407.227,369.717,174.440,43.053,158.494
C01519=1046.168,406.982,369.762,174.431,43.046,158.491
C01520=1046.159,406.736,369.807,174.423,43.038,158.489
C01521=1046.150,406.490,369.852,174.414,43.031,158.486
C01522=1046.140,406.245,369.897,174.405,43.025,158.484
C01523=1046.131,405.998,369.942,174.396,43.018,158.481
C01524=1046.122,405.755,369.986,174.387,43.011,158.479
C01525=1046.113,405.512,370.031,174.379,43.004,158.477
C01526=1046.103,405.269,370.075,174.370,42.998,158.474
C01527=1046.095,405.025,370.120,174.361,42.991,158.472
C01528=1046.086,404.783,370.163,174.353,42.984,158.469
C01529=1046.076,404.540,370.208,174.344,42.978,158.467
C01530=1046.067,404.296,370.252,174.336,42.971,158.465
C01531=1046.058,404.053,370.297,174.327,42.964,158.462
C01532=1046.049,403.808,370.340,174.319,42.957,158.460
C01533=1046.040,403.561,370.385,174.310,42.951,158.458
C01534=1046.030,403.316,370.430,174.302,42.944,158.455
C01535=1046.021,403.069,370.474,174.293,42.937,158.453
C01536=1046.012,402.823,370.519,174.285,42.931,158.451
C01537=1046.003,402.578,370.563,174.276,42.924,158.448
C01538=1045.994,402.332,370.607,174.268,42.918,158.446
C01539=1045.984,402.086,370.651,174.260,42.911,158.444
C01540=1045.976,401.840,370.695,174.252,42.904,158.441
C01541=1045.967,401.594,370.740,174.243,42.898,158.439
C01542=1045.958,401.348,370.784,174.235,42.891,158.437
C01543=1045.948,401.103,370.828,174.226,42.885,158.434
C01544=1045.939,400.857,370.873,174.218,42.879,158.432
C01545=1045.930,400.612,370.916,174.210,42.872,158.430
C01546=1045.921,400.365,370.960,174.201,42.865,158.428
C01547=1045.912,400.119,371.004,174.193,42.859,158.425
C01548=1045.903,399.873,371.048,174.185,42.853,158.423
C01549=1045.893,399.627,371.092,174.177,42.847,158.421
C01550=1045.885,399.382,371.135,174.169,42.840,158.419
C01551=1045.875,399.136,371.180,174.160,42.834,158.416
C01552=1045.867,398.889,371.223,174.153,42.827,158.414
C01553=1045.857,398.643,371.267,174.145,42.821,158.412
C01554=1045.849,398.398,371.310,174.136,42.815,158.410
C01555=1045.839,398.151,371.354,174.128,42.809,158.408
C01556=1045.831,397.906,371.398,174.120,42.802,158.405
C01557=1045.822,397.660,371.441,174.113,42.796,158.403
C01558=1045.813,397.414,371.485,174.104,42.790,158.401
C01559=1045.804,397.168,371.528,174.096,42.784,158.399
C01560=1045.795,396.922,371.571,174.089,42.777,158.397
C01561=1045.786,396.675,371.615,174.081,42.771,158.395
C01562=1045.778,396.430,371.659,174.072,42.765,158.392
C01563=1045.769,396.184,371.702,174.065,42.759,158.390
C01564=1045.760,395.938,371.745,174.057,42.753,158.388
C01565=1045.751,395.692,371.789,174.049,42.747,158.386
C01566=1045.742,395.446,371.831,174.042,42.741,158.384
C01567=1045.733,395.200,371.874,174.033,42.735,158.382
C01568=1045.724,394.954,371.918,174.026,42.729,158.380
C01569=1045.715,394.708,371.961,174.018,42.722,158.378
C01570=1045.707,394.462,372.004,174.010,42.716,158.376
C01571=1045.698,394.216,372.047,174.003,42.710,158.374
C01572=1045.689,393.970,372.090,173.995,42.705,158.371
C01573=1045.681,393.724,372.133,173.987,42.699,158.369
C01574=1045.672,393.478,372.176,173.979,42.693,158.367
C01575=1045.663,393.232,372.218,173.971,42.687,158.365
C01576=1045.654,392.985,372.262,173.964,42.681,158.363
C01577=1045.645,392.739,372.305,173.956,42.675,158.361
C01578=1045.637,392.493,372.348,173.949,42.669,158.359
C01579=1045.628,392.247,372.390,173.941,42.663,158.357
C01580=1045.619,392.001,372.432,173.934,42.657,158.355
C01581=1045.611,391.755,372.476,173.926,42.651,158.353
C01582=1045.602,391.509,372.518,173.919,42.646,158.351
C01583=1045.593,391.263,372.561,173.911,42.640,158.349
C01584=1045.580,390.879,372.626,173.899,42.631,158.346
C01585=1045.567,390.496,372.693,173.888,42.622,158.343
C01586=1045.553,390.113,372.759,173.877,42.613,158.340
C01587=1045.540,389.729,372.825,173.865,42.604,158.337
C01588=1045.531,389.484,372.867,173.858,42.599,158.335
C01589=1045.523,389.237,372.910,173.850,42.593,158.333
C01590=1045.514,388.991,372.951,173.843,42.587,158.331
C01591=1045.505,388.745,372.994,173.835,42.582,158.329
C01592=1045.496,388.498,373.036,173.828,42.576,158.327
C01593=1045.489,388.252,373.078,173.821,42.571,158.325
C01594=1045.479,388.006,373.121,173.814,42.565,158.323
C01595=1045.471,387.760,373.162,173.807,42.559,158.321
C01596=1045.462,387.513,373.205,173.800,42.554,158.320
C01597=1045.453,387.267,373.246,173.792,42.548,158.318
C01598=1045.444,387.021,373.288,173.785,42.543,158.316
C01599=1045.437,386.775,373.330,173.778,42.537,158.314
C01600=1045.428,386.528,373.372,173.770,42.532,158.312
C01601=1045.419,386.282,373.413,173.763,42.526,158.310
C01602=1045.411,386.035,373.456,173.757,42.521,158.309
C01603=1045.403,385.790,373.497,173.750,42.516,158.307
C01604=1045.394,385.543,373.539,173.742,42.510,158.305
C01605=1045.385,385.297,373.581,173.735,42.505,158.303
C01606=1045.377,385.051,373.622,173.728,42.499,158.301
C01607=1045.368,384.805,373.664,173.722,42.494,158.299
C01608=1045.360,384.558,373.706,173.714,42.489,158.297
C01609=1045.352,384.312,373.747,173.707,42.483,158.296
C01610=1045.343,384.065,373.789,173.700,42.478,158.294
C01611=1045.335,383.820,373.830,173.694,42.473,158.292
C01612=1045.327,383.572,373.872,173.686,42.467,158.290
C01613=1045.318,383.326,373.913,173.679,42.462,158.288
C01614=1045.309,383.080,373.955,173.672,42.457,158.287
C01615=1045.302,382.833,373.996,173.666,42.451,158.285
C01616=1045.293,382.587,374.038,173.659,42.446,158.283
C01617=1045.284,382.341,374.079,173.652,42.441,158.281
C01618=1045.276,382.095,374.120,173.645,42.436,158.279
C01619=1045.269,381.849,374.162,173.638,42.431,158.278
C01620=1045.260,381.602,374.203,173.631,42.425,158.276
C01621=1045.252,381.356,374.244,173.625,42.420,158.274
C01622=1045.243,381.109,374.285,173.618,42.415,158.272
C01623=1045.236,380.862,374.327,173.612,42.410,158.271
C01624=1045.227,380.616,374.368,173.604,42.405,158.269
C01625=1045.219,380.370,374.409,173.597,42.400,158.267
C01626=1045.211,380.124,374.450,173.591,42.394,158.265
C01627=1045.203,379.877,374.492,173.584,42.389,158.264
C01628=1045.195,379.631,374.533,173.578,42.384,158.262
C01629=1045.187,379.384,374.573,173.571,42.379,158.260
C01630=1045.178,379.137,374.614,173.564,42.374,158.259
C01631=1045.170,378.891,374.655,173.558,42.369,158.257
C01632=1045.162,378.645,374.695,173.551,42.364,158.255
C01633=1045.153,378.398,374.737,173.545,42.359,158.254
C01634=1045.145,378.152,374.778,173.538,42.354,158.252
C01635=1045.137,377.906,374.818,173.532,42.349,158.250
C01636=1045.129,377.658,374.859,173.524,42.344,158.248
C01637=1045.121,377.412,374.899,173.518,42.339,158.247
C01638=1045.113,377.166,374.940,173.512,42.334,158.245
C01639=1045.105,376.919,374.981,173.506,42.329,158.244
C01640=1045.093,376.569,375.038,173.496,42.322,158.241
C01641=1045.081,376.219,375.096,173.487,42.315,158.239
C01642=1045.069,375.870,375.154,173.477,42.308,158.237
C01643=1045.057,375.520,375.211,173.468,42.301,158.234
C01644=1045.050,375.273,375.251,173.462,42.296,158.233
C01645=1045.042,375.026,375.292,173.455,42.291,158.231
C01646=1045.033,374.780,375.332,173.449,42.287,158.229
C01647=1045.026,374.533,375.372,173.442,42.282,158.228
C01648=1045.018,374.287,375.413,173.436,42.277,158.226
C01649=1045.010,374.040,375.453,173.429,42.272,158.225
C01650=1045.001,373.794,375.493,173.424,42.268,158.223
C01651=1044.993,373.548,375.533,173.418,42.263,158.221
C01652=1044.986,373.301,375.573,173.411,42.258,158.220
C01653=1044.978,373.054,375.613,173.405,42.253,158.218
C01654=1044.970,372.808,375.654,173.399,42.248,158.217
C01655=1044.962,372.561,375.694,173.392,42.244,158.215
C01656=1044.954,372.315,375.734,173.386,42.239,158.213
C01657=1044.946,372.068,375.774,173.379,42.234,158.212
C01658=1044.938,371.821,375.814,173.373,42.230,158.210
C01659=1044.930,371.575,375.854,173.367,42.225,158.209
C01660=1044.922,371.328,375.894,173.361,42.220,158.207
C01661=1044.914,371.081,375.934,173.355,42.216,158.206
C01662=1044.906,370.835,375.975,173.349,42.211,158.204
C01663=1044.898,370.588,376.014,173.343,42.206,158.203
C01664=1044.890,370.341,376.054,173.336,42.202,158.201
C01665=1044.882,370.095,376.093,173.330,42.197,158.200
C01666=1044.874,369.848,376.133,173.324,42.192,158.198
C01667=1044.866,369.601,376.173,173.318,42.188,158.197
C01668=1044.858,369.354,376.212,173.312,42.184,158.195
C01669=1044.850,369.107,376.252,173.306,42.179,158.194
C01670=1044.842,368.861,376.291,173.299,42.175,158.192
C01671=1044.835,368.614,376.331,173.293,42.170,158.191
C01672=1044.826,368.368,376.371,173.288,42.166,158.189
C01673=1044.818,368.121,376.410,173.282,42.161,158.188
C01674=1044.810,367.874,376.449,173.275,42.156,158.186
C01675=1044.802,367.627,376.489,173.269,42.152,158.185
C01676=1044.795,367.381,376.528,173.264,42.148,158.183
C01677=1044.787,367.134,376.568,173.258,42.143,158.182
C01678=1044.778,366.887,376.607,173.252,42.139,158.180
C01679=1044.771,366.640,376.646,173.245,42.134,158.179
C01680=1044.764,366.394,376.686,173.240,42.130,158.177
C01681=1044.755,366.147,376.725,173.234,42.126,158.176
C01682=1044.748,365.900,376.764,173.228,42.121,158.174
C01683=1044.740,365.653,376.804,173.222,42.116,158.173
C01684=1044.732,365.407,376.843,173.217,42.112,158.172
C01685=1044.724,365.160,376.882,173.210,42.108,158.170
C01686=1044.717,364.913,376.922,173.204,42.104,158.169
C01687=1044.709,364.666,376.960,173.198,42.099,158.167
C01688=1044.701,364.419,377.000,173.193,42.094,158.166
C01689=1044.694,364.173,377.038,173.187,42.090,158.164
C01690=1044.686,363.926,377.078,173.181,42.086,158.163
C01691=1044.678,363.679,377.117,173.176,42.082,158.162
C01692=1044.671,363.432,377.156,173.170,42.077,158.160
C01693=1044.663,363.185,377.195,173.163,42.073,158.159
C01694=1044.656,362.939,377.235,173.158,42.069,158.157
C01695=1044.647,362.692,377.273,173.152,42.065,158.156
C01696=1044.638,362.362,377.325,173.145,42.059,158.154
C01697=1044.626,362.031,377.377,173.136,42.053,158.152
C01698=1044.617,361.701,377.429,173.129,42.048,158.150
C01699=1044.606,361.370,377.481,173.121,42.042,158.149
C01700=1044.598,361.123,377.519,173.115,42.038,158.147
C01701=1044.591,360.876,377.558,173.110,42.034,158.146
C01702=1044.583,360.629,377.596,173.104,42.030,158.144
C01703=1044.575,360.382,377.635,173.099,42.025,158.143
C01704=1044.567,360.136,377.673,173.093,42.021,158.142
C01705=1044.560,359.888,377.713,173.087,42.017,158.140
C01706=1044.552,359.642,377.751,173.082,42.013,158.139
C01707=1044.544,359.394,377.789,173.076,42.009,158.138
C01708=1044.537,359.148,377.828,173.071,42.005,158.137
C01709=1044.529,358.901,377.866,173.065,42.001,158.135
C01710=1044.521,358.654,377.904,173.059,41.997,158.134
C01711=1044.514,358.407,377.943,173.054,41.993,158.133
C01712=1044.506,358.160,377.982,173.048,41.989,158.131
C01713=1044.498,357.914,378.020,173.043,41.985,158.130
C01714=1044.491,357.667,378.058,173.037,41.981,158.129
C01715=1044.483,357.419,378.096,173.032,41.977,158.127
C01716=1044.476,357.173,378.135,173.026,41.973,158.126
C01717=1044.468,356.926,378.173,173.020,41.968,158.125
C01718=1044.461,356.678,378.211,173.016,41.964,158.123
C01719=1044.453,356.432,378.249,173.010,41.960,158.122
C01720=1044.445,356.185,378.287,173.005,41.957,158.121
C01721=1044.437,355.938,378.325,172.999,41.953,158.119
C01722=1044.430,355.691,378.363,172.994,41.948,158.118
C01723=1044.422,355.445,378.402,172.988,41.944,158.117
C01724=1044.414,355.197,378.439,172.983,41.941,158.116
C01725=1044.407,354.950,378.478,172.977,41.937,158.114
C01726=1044.399,354.703,378.515,172.972,41.933,158.113
C01727=1044.392,354.457,378.553,172.966,41.929,158.112
C01728=1044.384,354.209,378.591,172.961,41.925,158.110
C01729=1044.377,353.962,378.629,172.955,41.921,158.109
C01730=1044.369,353.715,378.667,172.951,41.917,158.108
C01731=1044.362,353.468,378.705,172.945,41.913,158.107
C01732=1044.354,353.221,378.743,172.940,41.910,158.106
C01733=1044.347,352.974,378.781,172.934,41.906,158.104
C01734=1044.339,352.726,378.818,172.929,41.902,158.103
C01735=1044.332,352.480,378.857,172.923,41.898,158.102
C01736=1044.325,352.233,378.894,172.919,41.894,158.101
C01737=1044.317,351.986,378.932,172.913,41.890,158.099
C01738=1044.310,351.738,378.969,172.908,41.887,158.098
C01739=1044.303,351.492,379.007,172.903,41.883,158.097
C01740=1044.295,351.245,379.044,172.897,41.879,158.096
C01741=1044.287,350.997,379.082,172.893,41.875,158.094
C01742=1044.279,350.750,379.120,172.887,41.871,158.093
C01743=1044.272,350.503,379.157,172.882,41.868,158.092
C01744=1044.265,350.256,379.195,172.876,41.864,158.091
C01745=1044.258,350.009,379.232,172.871,41.860,158.090
C01746=1044.250,349.762,379.269,172.867,41.857,158.088
C01747=1044.243,349.515,379.307,172.861,41.852,158.087
C01748=1044.235,349.268,379.344,172.856,41.849,158.086
C01749=1044.228,349.021,379.382,172.850,41.845,158.085
C01750=1044.220,348.774,379.419,172.845,41.842,158.084
C01751=1044.213,348.527,379.456,172.841,41.838,158.082
C01752=1044.203,348.202,379.505,172.834,41.833,158.081
C01753=1044.193,347.877,379.555,172.827,41.828,158.079
C01754=1044.183,347.552,379.603,172.820,41.823,158.078
C01755=1044.173,347.228,379.652,172.813,41.819,158.076
C01756=1044.166,346.981,379.689,172.808,41.815,158.075
C01757=1044.159,346.733,379.727,172.804,41.811,158.074
C01758=1044.151,346.487,379.763,172.798,41.808,158.073
C01759=1044.144,346.239,379.800,172.793,41.804,158.072
C01760=1044.137,345.992,379.838,172.789,41.801,158.070
C01761=1044.129,345.745,379.874,172.783,41.797,158.069
C01762=1044.122,345.498,379.911,172.778,41.794,158.068
C01763=1044.115,345.251,379.949,172.774,41.790,158.067
C01764=1044.107,345.003,379.985,172.768,41.786,158.066
C01765=1044.100,344.756,380.023,172.763,41.783,158.065
C01766=1044.092,344.509,380.059,172.758,41.779,158.064
C01767=1044.086,344.262,380.096,172.753,41.776,158.062
C01768=1044.078,344.015,380.133,172.748,41.772,158.061
C01769=1044.071,343.768,380.170,172.743,41.768,158.060
C01770=1044.064,343.520,380.207,172.738,41.765,158.059
C01771=1044.056,343.273,380.244,172.733,41.761,158.058
C01772=1044.049,343.026,380.280,172.729,41.758,158.057
C01773=1044.041,342.779,380.317,172.723,41.755,158.056
C01774=1044.035,342.531,380.354,172.719,41.751,158.054
C01775=1044.027,342.285,380.391,172.714,41.747,158.053
C01776=1044.020,342.038,380.427,172.708,41.744,158.052
C01777=1044.013,341.790,380.463,172.704,41.741,158.051
C01778=1044.006,341.542,380.500,172.699,41.737,158.050
C01779=1043.998,341.295,380.537,172.694,41.733,158.049
C01780=1043.990,341.048,380.573,172.689,41.730,158.048
C01781=1043.984,340.801,380.610,172.684,41.727,158.047
C01782=1043.976,340.554,380.646,172.680,41.723,158.046
C01783=1043.968,340.306,380.682,172.674,41.720,158.045
C01784=1043.961,340.060,380.719,172.670,41.717,158.044
C01785=1043.954,339.812,380.756,172.665,41.714,158.043
C01786=1043.946,339.565,380.792,172.660,41.710,158.041
C01787=1043.939,339.317,380.828,172.656,41.707,158.040
C01788=1043.932,339.070,380.864,172.650,41.703,158.039
C01789=1043.925,338.823,380.901,172.646,41.700,158.038
C01790=1043.917,338.576,380.937,172.641,41.697,158.037
C01791=1043.911,338.328,380.973,172.636,41.693,158.036
C01792=1043.903,338.081,381.010,172.631,41.690,158.035
C01793=1043.896,337.834,381.045,172.627,41.686,158.034
C01794=1043.888,337.587,381.082,172.622,41.683,158.033
C01795=1043.882,337.340,381.118,172.618,41.680,158.032
C01796=1043.874,337.092,381.154,172.612,41.677,158.031
C01797=1043.866,336.845,381.190,172.608,41.673,158.030
C01798=1043.860,336.598,381.227,172.603,41.670,158.029
C01799=1043.853,336.350,381.262,172.599,41.667,158.028
C01800=1043.846,336.103,381.298,172.593,41.663,158.026
C01801=1043.838,335.855,381.335,172.589,41.660,158.026
C01802=1043.832,335.608,381.371,172.584,41.657,158.025
C01803=1043.824,335.361,381.407,172.580,41.653,158.023
C01804=1043.817,335.114,381.442,172.575,41.650,158.022
C01805=1043.810,334.866,381.479,172.571,41.647,158.021
C01806=1043.802,334.619,381.514,172.565,41.644,158.020
C01807=1043.795,334.371,381.550,172.561,41.640,158.019
C01808=1043.785,334.043,381.598,172.555,41.636,158.018
C01809=1043.776,333.714,381.645,172.549,41.632,158.017
